ACTION A_DALICmdSetMinLevel_Input:
	IF emod = E_DALIAddressType.Group THEN
		byAddr		:= byGrpAdr;
		eAddrType	:= E_DALIAddressType.Group;
	ELSIF emod = E_DALIAddressType.Short THEN
		byAddr		:= byShrtAdr;
		eAddrType	:= E_DALIAddressType.Short;
	END_IF


	bActionBusy	:= TRUE;

	fbSetMinLevel(
		bError=> , 
		ipResultMessage=> , 
		bStart:= TRUE, 
		nAddress:= byAddr , 
		eAddressType:= eAddrType , 
		eCommandPriority:=Tc3_DALI.E_DALICommandPriority.Middle , 
		bBusy=> , 
		nMinLevel:= byDTR);
	

	IF (NOT fbSetMinLevel.bBusy) THEN
		IF fbSetMinLevel.bError THEN
			bErr := TRUE;
			nErrorId := fbSetMinLevel.ipResultMessage.nEventId;
		END_IF
		bActionBusy		:= FALSE;
		fbSetMinLevel(bStart:= FALSE);
	END_IF
END_ACTION

ACTION A_DALICmdStepDown:
	IF emod = E_DALIAddressType.Group THEN
		byAddr		:= byGrpAdr;
		eAddrType	:= E_DALIAddressType.Group;
	ELSIF emod = E_DALIAddressType.Short THEN
		byAddr		:= byShrtAdr;
		eAddrType	:= E_DALIAddressType.Short;
	END_IF

	bActionBusy	:= TRUE;

	fbStepDown(
		bError=> , 
		ipResultMessage=> , 
		bStart:= TRUE, 
		nAddress:=byAddr , 
		eAddressType:= eAddrType, 
		eCommandPriority:= E_DALICommandPriority.Middle, 
		bBusy=> );


	IF NOT fbStepDown.bBusy	THEN
		IF	fbStepDown.bError	THEN
			bErr     	:= TRUE;
		END_IF
		bActionBusy		:= FALSE;
		fbStepDown(bStart:= FALSE );
	END_IF
END_ACTION

ACTION A_DALICmdStepUp:
	IF emod = E_DALIAddressType.Group THEN
		byAddr		:= byGrpAdr;
		eAddrType	:= E_DALIAddressType.Group;
	ELSIF emod = E_DALIAddressType.Short THEN
		byAddr		:= byShrtAdr;
		eAddrType	:= E_DALIAddressType.Short;
	END_IF


	bActionBusy	:= TRUE;

	fbStepUp(
		bError=> , 
		ipResultMessage=> , 
		bStart:= TRUE, 
		nAddress:=byAddr , 
		eAddressType:=eAddrType , 
		eCommandPriority:= E_DALICommandPriority.Middle, 
		bBusy=> );


	IF NOT fbStepUp.bBusy	THEN
		IF	fbStepUp.bError	THEN
			bErr     	:= TRUE;
			nErrorId := fbStepUp.ipResultMessage.nEventId;

		END_IF
		bActionBusy		:= FALSE;
		fbStepUp(bStart:= FALSE);
	END_IF
END_ACTION

ACTION A_DALICmdUp:
	IF emod = E_DALIAddressType.Group THEN
		byAddr		:= byGrpAdr;
		eAddrType	:= E_DALIAddressType.Group;
	ELSIF emod = E_DALIAddressType.Short THEN
		byAddr		:= byShrtAdr;
		eAddrType	:= E_DALIAddressType.Short;
	END_IF

	bActionBusy	:= TRUE;

	fbUp(
		bError=> , 
		ipResultMessage=> , 
		bStart:= TRUE , 
		nAddress:=byAddr , 
		eAddressType:=eAddrType , 
		eCommandPriority:= E_DALICommandPriority.High, 
		bBusy=> );

	IF NOT fbUp.bBusy	THEN
		IF	fbUp.bError	THEN
			bErr     	:= TRUE;
			nErrorId := fbUp.ipResultMessage.nEventId;
		END_IF
		bActionBusy		:= FALSE;
		fbUp(bStart:= FALSE );
	END_IF
END_ACTION

ACTION A_ResetRoutine:
	tonSeqTimer(IN:=FALSE);
	tonDimRepeat(IN:=FALSE);

	bErr     	:= FALSE;
	nErrorId 	:= 0;


	fbUp						(bStart:= FALSE );
	fbDwn						(bStart:= FALSE );
	fbOff						(bStart:= FALSE );
	fbRecallMaxLevel			(bStart:= FALSE );
	fbRecallMinLevel			(bStart:= FALSE );
	fbDirectArcPowerControl		(bStart:= FALSE );
	fbStepUp					(bStart:= FALSE );
	fbStepDown					(bStart:= FALSE );
	fbQueryActualLevel			(bStart:= FALSE );
	fbSetFadeRate				(bStart:= FALSE );
	fbSetFadeTime				(bStart:= FALSE );
	fbQueryPhysicalMinLevel		(bStart:= FALSE );
	fbSetMinLevel				(bStart:= FALSE );
	fbQueryMinLevel				(bStart:= FALSE );
	fbSetMaxLevel				(bStart:= FALSE );
END_ACTION

{attribute 'monitoring' := 'call'}
PROPERTY ipDALICommunication : Tc3_DALI.I_DALICommunication
GET
ipDALICommunication := THIS^.ipCommunication;
END_GET
SET
THIS^.ipCommunicationPreset := ipDALICommunication;
END_SET
END_PROPERTY

//| Apply the perset value of IpCommunication if available
//| Return codes:
//|   FALSE: no peset value available
//|   TRUE: has taken the preset value
{attribute 'hide'}
METHOD PRIVATE TrySetCommunication : BOOL
VAR_INPUT
END_VAR
IF ((THIS^.ipCommunication <> THIS^.ipCommunicationPreset) AND (THIS^.ipCommunicationPreset <> 0)) THEN
	THIS^.ipCommunication := THIS^.ipCommunicationPreset;
	THIS^.fbUp.ipDALICommunication := THIS^.ipCommunication;
	THIS^.fbDwn.ipDALICommunication := THIS^.ipCommunication;
	THIS^.fbOff.ipDALICommunication := THIS^.ipCommunication;
	THIS^.fbRecallMaxLevel.ipDALICommunication := THIS^.ipCommunication;
	THIS^.fbRecallMinLevel.ipDALICommunication := THIS^.ipCommunication;
	THIS^.fbDirectArcPowerControl.ipDALICommunication := THIS^.ipCommunication;
	THIS^.fbStepUp.ipDALICommunication := THIS^.ipCommunication;	
	THIS^.fbStepDown.ipDALICommunication := THIS^.ipCommunication;
	THIS^.fbQueryActualLevel.ipDALICommunication := THIS^.ipCommunication;	
	THIS^.fbSetFadeRate.ipDALICommunication := THIS^.ipCommunication;
	THIS^.fbSetFadeTime.ipDALICommunication := THIS^.ipCommunication;
	THIS^.fbSetMaxLevel.ipDALICommunication := THIS^.ipCommunication;
	THIS^.fbSetMinLevel.ipDALICommunication := THIS^.ipCommunication;
	THIS^.fbQueryMinLevel.ipDALICommunication := THIS^.ipCommunication;	
	THIS^.fbQueryMaxLevel.ipDALICommunication := THIS^.ipCommunication;
	THIS^.fbQueryPhysicalMinLevel.ipDALICommunication := THIS^.ipCommunication;
	THIS^.fbQueryActualLevelBackgound.ipDALICommunication := THIS^.ipCommunication;
	THIS^.fbQueryStatusBackground.ipDALICommunication := THIS^.ipCommunication;
	TrySetCommunication := TRUE;
ELSE
	TrySetCommunication := FALSE;
END_IF
END_METHOD

END_FUNCTION_BLOCK

// POUs/DALI/Operators/FB_BA_ValTrigF
///Trigger-setting of a value, when it leaves a specific hysteresis
FUNCTION_BLOCK FB_BA_ValTrigF
VAR_INPUT
	bEn			: BOOL;		(* Enable *)
	bRetrig		: BOOL;		(* Retrigger - send bSet for one cycle *)
	fIn		: REAL;	(* Input signal *)
	fHys		: REAL;	(* Signal Hysteresis *)
END_VAR
VAR_OUTPUT
	fOut		: REAL;
	bSet		: BOOL;
END_VAR
VAR
	bInit		: BOOL;
	rtRetrig1	: R_TRIG;
	rtRetrig2	: R_TRIG;
	fLimUp		: REAL;
	fLimDwn		: REAL;
	uiStep		: UINT;
END_VAR

IF NOT bInit	THEN
	fLimUp	:= fIn+fHys/2;
	fLimDwn:= fIn-fHys/2;
	fOut	:= fIn;
	bInit	:= TRUE;
END_IF

rtRetrig1(CLK:=bEn); 		(*Retrigger both at retrigger-command and at beginning of enable*)
rtRetrig2(CLK:=bRetrig); (*Retrigger both at retrigger-command and at beginning of enable*)

CASE uiStep OF
0: (*Idle*)
	bSet:=FALSE;
	IF (fIn>=fLimUp)OR(fIn<=fLimDwn) OR rtRetrig1.Q	OR rtRetrig2.Q	THEN
		uiStep	:= 10;
	END_IF
	IF NOT bEn	THEN
		uiStep	:= 0;
	END_IF

10:
	fLimUp	:= fIn+fHys/2;
	fLimDwn	:= fIn-fHys/2;
	fOut	:= fIn;
	bSet	:= TRUE;
	uiStep 	:= 0;
END_CASE

END_FUNCTION_BLOCK

// POUs/DALI/Ballast/FB_DALILgtActr_Simple
FUNCTION_BLOCK FB_DALILgtActr_Simple  (* V1.1 dfgdfgdfgdfgdfgfzxcv *)
VAR_INPUT
	byShrtAdr				: BYTE;
	byGrpAdr				: BYTE;
	eMod					: E_DALIAddressType:= E_DALIAddressType.Group;
	fSttupCtrlVal			: REAL;
	fLgtOffset				: REAL;
	uiBlinkTi				: UINT;
	uiOffDly				: UINT;
	uiPollActLgtLvl			: UINT;
	bReInit					: BOOL;
	stLgtCmd				: ST_LgtCmd;
	DALI_LINE_NUM			: BYTE;
END_VAR
VAR_OUTPUT
	fActlLgtLvl				: REAL;
	byActlLgtLvl			: BYTE;
	bLgt					: BOOL;
	fActlMinCtrlVal			: REAL;
	bMinCtrlValRchd 		: BOOL;
	fActlMaxCtrlVal			: REAL;
	bMaxCtrlValRchd 		: BOOL;
	fRstVal					: REAL;
	eActlFadeTime			: E_DALIFadeTime;
	eActlFadeRate			: E_DALIFadeRate;
	byPhysMinVal			: BYTE;
	byActlMinCtrlVal		: BYTE;
	byActlMaxCtrlVal		: BYTE;
	bInitDevice				: BOOL;
	bBlinkSeqStarted 		: BOOL;
	bActionBusy				: BOOL;
	bErr     				: BOOL;
	nErrorId				: UDINT;
	byDALIDevSta			: BYTE;
END_VAR
VAR
	ipCommunication					: I_DALICommunication;
	ipCommunicationPreset			: I_DALICommunication;

	bInit					: BOOL;
	bBusy					: BOOL;
	bRstErr					: BOOL;
	rtReInit				: R_TRIG;
	bReactCmdSt				: BOOL;
	byAddr					: BYTE;
	eAddrType				: E_DALIAddressType;
	byArcPowerLevel			: BYTE;
	byDTR					: BYTE;
	uiCmdStep				: UINT;

	bDimUp					: BOOL;
	bDimDwn					: BOOL;
	bSetMinValInput			: BOOL;	(*Änderung MinVal über Bausteineingang*)
	bSetMaxValInput			: BOOL;	(*Änderung MaxVal über Bausteineingang*)
	bySetMinValInput		: BYTE;
	bySetMaxValInput		: BYTE;
	bSetMinValCmdSt			: BOOL;	(*Änderung MinVal über Kommandostruktur*)
	bSetMaxValCmdSt			: BOOL;	(*Änderung MaxVal über Kommandostruktur*)
	bySetMinValCmdSt		: BYTE;
	bySetMaxValCmdSt		: BYTE;
	byRstVal				: BYTE;
	bySttupCtrlVal			: BYTE;
	rtInitDevice			: R_TRIG;
	rtOff					: R_TRIG;
	rtClMinCtrlVal			: R_TRIG;
	rtClMaxCtrlVal			: R_TRIG;
	rtClOnVal				: R_TRIG;
	rtClRstVal				: R_TRIG;
	rtSetCtrlValDct			: R_TRIG;
	rtChgMaxCtrlVal			: R_TRIG;
	rtChgMinCtrlVal			: R_TRIG;
	rtStpUp							: R_TRIG;
	rtStpDwn						: R_TRIG;
	rtRmp							: R_TRIG;
	tonSeqTimer						: TON;
	tonDimRepeat					: TON;
	fbUp							: FB_DALI102Up(0);
	fbDwn							: FB_DALI102Down(0);
	fbOff							: FB_DALI102Off(0);
	fbRecallMaxLevel				: FB_DALI102RecallMaxLevel(0);
	fbRecallMinLevel				: FB_DALI102RecallMinLevel(0);
	fbDirectArcPowerControl			: FB_DALI102DirectArcPowerControl(0);
	fbStepUp						: FB_DALI102StepUp(0);
	fbStepDown						: FB_DALI102StepDown(0);
	fbQueryActualLevel				: FB_DALI102QueryActualLevel(0);
	fbQueryMinLevel					: FB_DALI102QueryMinLevel(0);
	fbQueryMaxLevel					: FB_DALI102QueryMaxLevel(0);
	fbQueryPhysicalMinLevel			: FB_DALI102QueryPhysicalMinimum(0);
	fbQueryActualLevelBackgound		: FB_DALI102QueryActualLevel(0);
	fbQueryStatusBackground			: FB_DALI102QueryStatus(0);
	fbSendValue						: FB_BA_ValTrigf;
	fbReTrigSend0					: R_TRIG;
	nStepQueryActualLevel			: UINT;
	tonCycleActualLevelMasterDev	: TON;
	bSetRetry						: BOOL;
	fbTimeOut						: TON;
	byActlFadeTime					: BYTE;
	fbGETCURTASKINDEX				: GETCURTASKINDEX;
	nCurrentIdx						: BYTE;
	nCycleTimeInMS					: UDINT;
	nCycleCountSP					: UDINT;
	nActualCount					: UDINT:= 1;
END_VAR
VAR_IN_OUT
END_VAR



(* For checking which task the FB are called*)
fbGETCURTASKINDEX(index=>nCurrentIdx );
nCycleTimeInMS:= (_TaskInfo[nCurrentIdx].CycleTime/10000);
IF nCycleTimeInMS > 0 THEN	(*nCycleCountSP are only calculated if nCycleTimeInMS are larger than 0*)
	nCycleCountSP:= (200 / nCycleTimeInMS) ; (* 200 are the target time between 2 UP/Down cmd*)
END_IF

{region "initialize the outputs"}
IF (NOT bInit) THEN
	THIS^.TrySetCommunication();		 
	bBusy := TRUE;
	nErrorId := 0;
	bErr := FALSE;
	bInit := TRUE;
END_IF
{endregion}


{region "check parameters"}
IF (ipCommunication = 0) THEN
	bErr := TRUE;
	nErrorId := TC_EVENTS.TcDALIEventClass.TheInterfaceToTheCommunicationBufferIsNotInitialized.nEventId;
	uiCmdStep := 0;
END_IF
IF ((eMod <> E_DALIAddressType.Short) AND (eMod <> E_DALIAddressType.Group) AND (eMod <> E_DALIAddressType.Broadcast) AND (eMod <> E_DALIAddressType.BroadcastUnaddr)) THEN
	bErr := TRUE;
	nErrorId := TC_EVENTS.TcDALIEventClass.ParameterAddressTypeLiesOutsideOfTheValidRange.nEventId;
	uiCmdStep := 0;
END_IF
IF ((eMod = E_DALIAddressType.Short) AND (byShrtAdr > 63)) THEN
	bErr := TRUE;
	nErrorId := TC_EVENTS.TcDALIEventClass.ParameterAddressIsAShortAddressAndLiesOutsideOfTheValidRange.nEventId;
	uiCmdStep := 0;
END_IF
IF ((eMod = E_DALIAddressType.Group) AND (byGrpAdr > 15)) THEN
	bErr := TRUE;
	nErrorId := TC_EVENTS.TcDALIEventClass.ParameterAddressIsAGroupAddressAndLiesOutsideOfTheValidRange.nEventId;
	uiCmdStep := 0;
END_IF
IF (byShrtAdr > 63) THEN
	bErr := TRUE;
	nErrorId := 16#8000; // custom error code: Parameter byShrtAdr lies outside of the valid range
	uiCmdStep := 0;
END_IF
	
IF (byGrpAdr > 15) THEN
	bErr := TRUE;
	nErrorId := 16#8001; // custom error code: Parameter byGrpAdr lies outside of the valid range
	uiCmdStep := 0;
END_IF
{endregion}

(*	bRstErr ist ein Fehlermerker: wenn vorher über Fehler, s.o. herausgesprungen wurde und nun "alles gut" ist,
dann hier Fehler einmalig zurücksetzen, damit im weiteren Verlauf die Warnmeldungen sichtbar werden können*)
IF	bRstErr  THEN
		bRstErr    	:= FALSE;
		bErr     	:= FALSE;
END_IF


(* + + + + + + + + + + + + + + + + + + + + + + + + + + + + + + + + + + + + + + + + + + + + *)
(*In den DALI-Ausführungsaktionen ist jedoch zur Sicherheit noch ein RETURN-Aussprung*)
IF (eMod=E_DALIAddressType.Short)	THEN
	bReactCmdSt:=FALSE;
ELSE
	bReactCmdSt:=TRUE;
END_IF

(* + + + + + + + + + + + + + + + + + + + + + + + + + + + + + + + + + + + + + + + + + + + + *)
(*Init *)
rtReInit	 (CLK:=bReInit);
IF bReInit	THEN
	bInit:=FALSE;
END_IF

IF NOT bInit	THEN
	rtInitDevice			(CLK:=FALSE);
	bInitDevice			:= TRUE;

	bInit					:= TRUE;
	tonDimRepeat		(PT:=t#200ms);

	IF fSttupCtrlVal < 0.0	 THEN
		bySttupCtrlVal	:= 0;
	ELSIF	fSttupCtrlVal > 100.0	 THEN
		bySttupCtrlVal	:= 254;
	ELSE
		bySttupCtrlVal	:= LREAL_TO_BYTE(F_fDALICurve(fSttupCtrlVal));
	END_IF
END_IF

rtInitDevice (CLK:=bInitDevice);

(*Removed in Simple version, Other FB needed for setup ballast - HMB 14/12-2021*)
(*

(* + + + + + + + + + + + + + + + + + + + + + + + + + + + + + + + + + + + + + + + + + + + + *)
(*Change DimTime/FadeRate über Bausteineingang*)
IF	(uiDimTi<>uiDimTi_SV) OR rtInitDevice.Q THEN
	A_DimTimeToFadeRate;
	uiDimTi_SV	:= uiDimTi;
	IF NOT rtInitDevice.Q	THEN
		bSetFadeRate	:= TRUE;
	END_IF
END_IF

(* + + + + + + + + + + + + + + + + + + + + + + + + + + + + + + + + + + + + + + + + + + + + *)
(*Change Min-/MaxCtrlVal über Bausteineingang*)

IF	(lrMinCtrlVal<>lrMinCtrlVal_SV) OR rtInitDevice.Q THEN
	lrMinCtrlVal_SV		:= lrMinCtrlVal;
	IF 		lrMinCtrlVal < 0.0		 THEN
		bySetMinValInput	:= 0;
	ELSIF	lrMinCtrlVal > 100.0	 THEN
		bySetMinValInput	:= 254;
	ELSE
		bySetMinValInput	:= LREAL_TO_BYTE(lrMinCtrlVal*2.54);
	END_IF
	IF NOT rtInitDevice.Q	THEN
		bSetMinValInput	:= TRUE;
	END_IF
END_IF

IF	(lrMaxCtrlVal<>lrMaxCtrlVal_SV) OR rtInitDevice.Q THEN
	lrMaxCtrlVal_SV		:= lrMaxCtrlVal;
	IF 		lrMaxCtrlVal < 0.0		 THEN
		bySetMaxValInput	:= 0;
	ELSIF	lrMaxCtrlVal > 100.0	 THEN
		bySetMaxValInput	:= 254;
	ELSE
		bySetMaxValInput	:= LREAL_TO_BYTE(lrMaxCtrlVal*2.54);
	END_IF
	IF NOT rtInitDevice.Q	THEN
		bSetMaxValInput	:= TRUE;
	END_IF
END_IF


(* + + + + + + + + + + + + + + + + + + + + + + + + + + + + + + + + + + + + + + + + + + + + *)
(*Change Min-/MaxCtrlVal über Kommandostruktur*)
rtChgMinCtrlVal	(CLK:= stLgtCmd.bChgMinCtrlVal);
rtChgMaxCtrlVal	(CLK:= stLgtCmd.bChgMaxCtrlVal);

IF 	rtChgMinCtrlVal.Q	AND bReactCmdSt			THEN
	IF 		stLgtCmd.lrChgMinCtrlVal < 0.0		 THEN
		bySetMinValCmdSt	:= 0;
	ELSIF	stLgtCmd.lrChgMinCtrlVal > 100.0	 THEN
		bySetMinValCmdSt	:= 254;
	ELSE
		bySetMinValCmdSt	:= LREAL_TO_BYTE(stLgtCmd.lrChgMinCtrlVal*2.54);
	END_IF
	bSetMinValCmdSt	:= TRUE;
END_IF

IF 	rtChgMaxCtrlVal.Q	AND bReactCmdSt			THEN
	IF 		stLgtCmd.lrChgMaxCtrlVal < 0.0		 THEN
		bySetMaxValCmdSt	:= 0;
	ELSIF	stLgtCmd.lrChgMaxCtrlVal > 100.0	 THEN
		bySetMaxValCmdSt	:= 254;
	ELSE
		bySetMaxValCmdSt	:= LREAL_TO_BYTE(stLgtCmd.lrChgMaxCtrlVal*2.54);
	END_IF
	bSetMaxValCmdSt	:= TRUE;
END_IF
*)

fbSendValue(bEn:= TRUE, bRetrig:= , fIn:= stLgtCmd.fSetCtrlValDct, fHys:= 0.1);

IF bMinCtrlValRchd AND stLgtCmd.fSetCtrlValDct = 0 THEN
	fbReTrigSend0(CLK:=TRUE , Q=> );
ELSE
	fbReTrigSend0(CLK:=FALSE , Q=> );
END_IF

(* + + + + + + + + + + + + + + + + + + + + + + + + + + + + + + + + + + + + + + + + + + + + *)
(* Flankenbildung und Verriegelung der Schalt- und Dimmbefehle *)
rtOff			(CLK:=stLgtCmd.bOff OR fbReTrigSend0.Q);
rtClMinCtrlVal	(CLK:=stLgtCmd.bClMinCtrlVal);
rtClMaxCtrlVal	(CLK:=stLgtCmd.bClMaxCtrlVal);
rtClOnVal		(CLK:=stLgtCmd.bClOnVal);
rtClRstVal		(CLK:=stLgtCmd.bClRstVal);
rtSetCtrlValDct	(CLK:=stLgtCmd.bSetCtrlValDct OR fbSendValue.bSet);
rtStpUp			(CLK:=stLgtCmd.bStpUp);
rtStpDwn		(CLK:=stLgtCmd.bStpDwn);

bDimUp			:= stLgtCmd.bDimUp;
bDimDwn			:= stLgtCmd.bDimDwn;

(* + + + + + + + + + + + + + + + + + + + + + + + + + + + + + + + + + + + + + + + + + + + + *)
(* Priorisierung aller Befehle und Schrittzuweisung *)
IF NOT bBusy	THEN
	IF			rtInitDevice.Q		THEN
				bBusy := TRUE;
								A_ResetRoutine();
				uiCmdStep:=1030;	(*Jump over write to ballast, else set back to step 1000*)
	ELSIF	bDimUp				AND NOT bMaxCtrlValRchd THEN
				bBusy := TRUE;
				A_ResetRoutine();
				uiCmdStep:=10;
	ELSIF	bDimDwn				AND NOT bMinCtrlValRchd THEN
				bBusy := TRUE;
				A_ResetRoutine();
				uiCmdStep:=20;
	ELSIF	rtOff.Q				THEN
				bBusy := TRUE;
				A_ResetRoutine();
				uiCmdStep:=30;
	ELSIF	rtClMinCtrlVal.Q	THEN
				bBusy := TRUE;
				A_ResetRoutine();
				uiCmdStep:=40;
	ELSIF	rtClMaxCtrlVal.Q	THEN
				bBusy := TRUE;
				A_ResetRoutine();
				uiCmdStep:=50;
	ELSIF	rtClOnVal.Q	THEN
				bBusy := TRUE;
				A_ResetRoutine();
				uiCmdStep:=60;
	ELSIF	rtClRstVal.Q		THEN
				bBusy := TRUE;
				A_ResetRoutine();
				uiCmdStep:=70;
	ELSIF	rtSetCtrlValDct.Q	THEN
				bBusy := TRUE;
				A_ResetRoutine();
				uiCmdStep:=80;
	ELSIF	rtStpUp.Q			AND NOT bMaxCtrlValRchd THEN
				bBusy := TRUE;
				A_ResetRoutine();
				uiCmdStep:=90;
	ELSIF	rtStpDwn.Q			AND NOT bMinCtrlValRchd THEN
				bBusy := TRUE;
				A_ResetRoutine();
				uiCmdStep:=100;
	END_IF
END_IF

(* + + + + + + + + + + + + + + + + + + + + + + + + + + + + + + + + + + + + + + + + + + + + *)
(*Kommandoausgabe*)
CASE uiCmdStep OF

0: (*Idle*)
	bInitDevice := FALSE;
	bBusy := FALSE;


(* - - - - - - - - - - - - - - - - - - - - - - - - *)
10:(*Dim Up*)
	bBlinkSeqStarted := FALSE;
(*	tonDimRepeat	(IN:=TRUE); *)  (*Disabled for at teste om Up cmd kommer hurtigere ved at tælle skan, istedet for timer*)
	nActualCount:= 1;
		A_DALICmdUp();
	IF NOT bActionBusy	THEN
		uiCmdStep:= 11;
	END_IF

11:(*Ende Wartezeit 200ms abwarten*)

(*Disablet to be more precise in case of long scantimes in the task - HMB 13/12-2021*)
(*	tonDimRepeat();
	IF tonDimRepeat.Q THEN
		tonDimRepeat(IN:= FALSE);
		IF bDimUp		THEN
			uiCmdStep:=10;
		ELSE
			uiCmdStep:=12;
		END_IF
	END_IF
*)
	(* Added to see if 200ms can be reached with this scan count*)
	IF nActualCount <= nCycleCountSP THEN
		nActualCount := nActualCount + 1;
		IF nActualCount >=nCycleCountSP THEN
			nActualCount:=1;
			IF bDimUp		THEN
				uiCmdStep:=10;
			ELSE
				uiCmdStep:=12;
			END_IF
		END_IF
	END_IF


12: (*Lichtabfrage wenn fertig*)
		A_DALICmdQueryActualLevel();
	IF NOT bActionBusy	THEN
		byActlLgtLvl	:= fbQueryActualLevel.nActualLevel;
		uiCmdStep		:= 0;
	END_IF

(* - - - - - - - - - - - - - - - - - - - - - - - - *)
20:(*Dim Down*)
	bBlinkSeqStarted := FALSE;
(*	tonDimRepeat	(IN:=TRUE); *)  (*Disabled for at teste om Up cmd kommer hurtigere ved at tælle skan, istedet for timer*)
	nActualCount:= 1;
		A_DALICmdDown();
	IF NOT bActionBusy	THEN
		uiCmdStep:= 21;
	END_IF

21:(*Ende Wartezeit 200ms abwarten*)
(*Disablet to be more precise in case of long scantimes in the task - HMB 13/12-2021*)
(*	tonDimRepeat();
	IF tonDimRepeat.Q THEN
		tonDimRepeat(IN:= FALSE);
		IF bDimDwn		THEN
			uiCmdStep:=20;
		ELSE
			uiCmdStep:=22;
		END_IF
	END_IF
*)
	IF nActualCount <= nCycleCountSP THEN
		nActualCount := nActualCount + 1;
		IF nActualCount >=nCycleCountSP THEN
			nActualCount:= 1;
			IF bDimDwn	THEN
				uiCmdStep:=20;
			ELSE
				uiCmdStep:=22;
			END_IF
		END_IF
	END_IF

22: (*Lichtabfrage wenn fertig*)
		A_DALICmdQueryActualLevel();
	IF NOT bActionBusy	THEN
		byActlLgtLvl	:= fbQueryActualLevel.nActualLevel;
		uiCmdStep		:= 0;
	END_IF

(* - - - - - - - - - - - - - - - - - - - - - - - - *)
30:(*Off*)
		A_DALICmdOff();
	IF NOT bActionBusy	THEN
		byActlLgtLvl	:=0;
		IF (uiOffDly<>0) AND NOT bBlinkSeqStarted AND NOT bErr	THEN
			uiCmdStep:=500;
		ELSE
			bBlinkSeqStarted := FALSE;
			uiCmdStep:= 0;
		END_IF
	END_IF

(* - - - - - - - - - - - - - - - - - - - - - - - - *)
40:(*Call MinCtrlVal*)
	bBlinkSeqStarted := FALSE;
		A_DALICmdRecallMinLevel();
	IF NOT bActionBusy	THEN
		byActlLgtLvl:=byActlMinCtrlVal;
		uiCmdStep:= 0;
	END_IF

(* - - - - - - - - - - - - - - - - - - - - - - - - *)
50:(*Call MaxCtrlVal*)
	bBlinkSeqStarted := FALSE;
		A_DALICmdRecallMaxLevel();
	IF NOT bActionBusy	THEN
		byActlLgtLvl:=byActlMaxCtrlVal;
		uiCmdStep:= 0;
	END_IF

(* - - - - - - - - - - - - - - - - - - - - - - - - *)
60:(*Call OnVal*)
	(*Limitation is not to be left to the electrical device -> the output of the actual value would be left to the background-polling only*)
	IF ((stLgtCmd.lrOnVal)>=fActlMaxCtrlVal)	THEN
		byArcPowerLevel:=byActlMaxCtrlVal;
	ELSIF ((stLgtCmd.lrOnVal)<=0.0)	THEN
		byArcPowerLevel:=0;
	ELSIF ((stLgtCmd.lrOnVal)<=fActlMinCtrlVal)	THEN
		byArcPowerLevel:=byActlMinCtrlVal;
	ELSE
		byArcPowerLevel:=LREAL_TO_BYTE((stLgtCmd.lrOnVal)*2.54);
	END_IF

		A_DALICmdDirectArcPowerControl();
	IF NOT bActionBusy	THEN
		byActlLgtLvl:=byRstVal;
		uiCmdStep:= 0;
	END_IF

(* - - - - - - - - - - - - - - - - - - - - - - - - *)
70:(*Call ResetVal*)
	bBlinkSeqStarted := FALSE;
	byArcPowerLevel	:= byRstVal;
		A_DALICmdDirectArcPowerControl();
	IF NOT bActionBusy	THEN
		byActlLgtLvl:=byRstVal;
		uiCmdStep:= 0;
	END_IF

(* - - - - - - - - - - - - - - - - - - - - - - - - *)
80:(*Set Control value directly*)
	(*Limitation is not to be left to the electrical device -> the output of the actual value would be left to the background-polling only*)
	byArcPowerLevel:= LIMIT(0,LREAL_TO_BYTE(F_fDALICurve(stLgtCmd.fSetCtrlValDct+ fLgtOffset)),254);
	A_DALICmdDirectArcPowerControl();
	IF NOT bActionBusy	THEN
(*		byActlLgtLvl:=byArcPowerLevel;*)
		IF (byActlLgtLvl=0) AND (uiOffDly<>0) AND NOT bBlinkSeqStarted AND NOT bErr	THEN
			uiCmdStep:=500;
		ELSE
			bBlinkSeqStarted := FALSE;
			uiCmdStep:= 0;
		END_IF
	END_IF

(* - - - - - - - - - - - - - - - - - - - - - - - - *)
90:(*Step Up*)
	bBlinkSeqStarted := FALSE;
		A_DALICmdStepUp();
	IF NOT bActionBusy	THEN
		byActlLgtLvl:=byActlLgtLvl+1;
		IF	byActlLgtLvl>byActlMaxCtrlVal	THEN
			byActlLgtLvl:=byActlMaxCtrlVal;
		END_IF
		uiCmdStep:= 0;
	END_IF

(* - - - - - - - - - - - - - - - - - - - - - - - - *)
100:(*Step Down*)
	bBlinkSeqStarted := FALSE;
		A_DALICmdStepDown();
	IF NOT bActionBusy	THEN
		byActlLgtLvl:=byActlLgtLvl-1;
		IF	byActlLgtLvl<byActlMinCtrlVal	THEN
			byActlLgtLvl:=byActlMinCtrlVal;
		END_IF
		uiCmdStep:= 0;
	END_IF


(* - - - - - - - - - - - - - - - - - - - - - - - - *)
(*ZUR SICHERHEIT: ABFRAGE NACH PARAMETRIERUNG*)
350:(*Query Min Level*)
	A_DALICmdQueryMinLevel();
	IF NOT bActionBusy	THEN
		IF bErr	THEN
			uiCmdStep:= 0;
		ELSE
			uiCmdStep:= 351;
		END_IF
	END_IF
	byActlMinCtrlVal:=fbQueryMinLevel.nMinLevel;
	fActlMinCtrlVal := LIMIT(0,LREAL_TO_BYTE(F_fDALICurve(byActlMinCtrlVal)), 254);

351:(*Query Max Level*)
	A_DALICmdQueryMaxLevel();
	IF NOT bActionBusy	THEN
		IF bErr	THEN
			uiCmdStep:= 0;
		ELSE
			uiCmdStep:= 352;
		END_IF
	END_IF
	byActlMaxCtrlVal:=fbQueryMaxLevel.nMaxLevel;
	fActlMaxCtrlVal := LIMIT(0,LREAL_TO_BYTE(F_fDALICurve(byActlMaxCtrlVal)), 254);

352: (*Lichtabfrage wenn fertig*)
		A_DALICmdQueryActualLevel();
	IF NOT bActionBusy	THEN
		byActlLgtLvl	:= fbQueryActualLevel.nActualLevel;
		uiCmdStep		:= 0;
	END_IF


(* - - - - - - - - - - - - - - - - - - - - - - - - *)
(*Ausschalt-Blinksequenz*)
500: (*Lampe ist bereits aus -> Wartezeit Blinktime*)
	bBusy				:= FALSE;	(*Blinksequenz soll unterbrechbar sein*)
	bBlinkSeqStarted	:= TRUE;
	tonSeqTimer			(IN:= TRUE, PT:=UDINT_TO_TIME(uiBlinkTi*1000));

	IF tonSeqTimer.Q	THEN
		bBusy := TRUE;	(*Verriegelung Kommandoannahme*)
		tonSeqTimer(IN:=FALSE);
		uiCmdStep:= 505;
	END_IF

505: (*Zurück auf ürsprünglich gespeicherten Wert*)
	byArcPowerLevel	:= byRstVal;
		A_DALICmdDirectArcPowerControl();
	IF NOT bActionBusy	THEN
		byActlLgtLvl := byRstVal;
		bBusy:= FALSE;	(*Blinksequenz soll wieder unterbrechbar sein*)
		IF bErr	THEN
			uiCmdStep:= 0;
		ELSE
			uiCmdStep:= 510;
		END_IF
	END_IF

510:(*Wartezeit Off-Delaytime*)
	tonSeqTimer(IN:= TRUE, PT:=UDINT_TO_TIME(uiOffDly*1000));
	IF tonSeqTimer.Q THEN
		bBusy := TRUE;	(*Verriegelung Kommandoannahme*)
		tonSeqTimer(IN:=FALSE);
		uiCmdStep:= 515;
	END_IF

515:(*Off*)
		A_DALICmdOff();
	IF NOT bActionBusy	THEN
		byActlLgtLvl		:= 0;
		bBlinkSeqStarted	:= FALSE;
		bBusy				:= FALSE;
		uiCmdStep			:= 0;
	END_IF

(* - - - - - - - - - - - - - - - - - - - - - - - - *)
(*Init Device-Routine*)

1000: (*Wait fort free DT8*)
	IF NOT arrbBlockDTR[DALI_LINE_NUM] THEN
		uiCmdStep:= 1030;
		arrbBlockDTR[DALI_LINE_NUM]:= FALSE;
	END_IF


1030:(*Query physical Min Level*)
		A_DALICmdQueryPhysicalMinLevel();
	IF NOT bActionBusy	THEN
		IF bErr	THEN
			uiCmdStep:= 0;
			arrbBlockDTR[DALI_LINE_NUM]:=FALSE;
		ELSE
			uiCmdStep:= 1035;
		END_IF
	END_IF
	byPhysMinVal:=fbQueryPhysicalMinLevel.nPhysicalMinimum;

1035:(*Query Min Level*)
		A_DALICmdQueryMinLevel();
	IF NOT bActionBusy	THEN
		IF bErr	THEN
			uiCmdStep:= 0;
			arrbBlockDTR[DALI_LINE_NUM]:=FALSE;
		ELSE
			uiCmdStep:= 1040;
		END_IF
	END_IF
	byActlMinCtrlVal:=fbQueryMinLevel.nMinLevel;
	fActlMinCtrlVal := LIMIT(0,LREAL_TO_BYTE(F_fDALICurve(byActlMinCtrlVal)), 254);

1040:(*Query Max Level*)
		A_DALICmdQueryMaxLevel();
	IF NOT bActionBusy	THEN
		IF bErr	THEN
			uiCmdStep:= 0;
			arrbBlockDTR[DALI_LINE_NUM]:=FALSE;
		ELSE
			uiCmdStep:= 1045;
		END_IF
	END_IF
	byActlMaxCtrlVal:=fbQueryMaxLevel.nMaxLevel;
	fActlMaxCtrlVal := LIMIT(0,LREAL_TO_BYTE(F_fDALICurve(byActlMaxCtrlVal)), 254);

1045:(*Call Startup-Level*)
	byArcPowerLevel	:= bySttupCtrlVal;
		A_DALICmdDirectArcPowerControl_Sttup();
	IF NOT bActionBusy	THEN
		uiCmdStep:= 1050;
	END_IF

1050: (*Lichtabfrage wenn fertig*)
		A_DALICmdQueryActualLevel();
	IF NOT bActionBusy	THEN
		byActlLgtLvl	:= fbQueryActualLevel.nActualLevel;
		uiCmdStep		:= 0;
		arrbBlockDTR[DALI_LINE_NUM]:=FALSE;
	END_IF

END_CASE

(*+ + + + + + + + + + + + + + + + + + + + + + + + + + + + + + + + + + + + + + + + + + + + + + + + +*)

IF ((uiPollActLgtLvl > 0) AND (nStepQueryActualLevel = 0) AND (bErr = FALSE)) THEN
	tonCycleActualLevelMasterDev(IN := TRUE, PT := UINT_TO_TIME(uiPollActLgtLvl*1000));
	IF (tonCycleActualLevelMasterDev.Q) THEN
		tonCycleActualLevelMasterDev(IN := FALSE);
		nStepQueryActualLevel := 10;
	END_IF
END_IF

CASE nStepQueryActualLevel OF
0:
	;
10:
	fbQueryActualLevelBackgound(
		bError=> , 
		ipResultMessage=> , 
		bStart:= TRUE, 
		nAddress:= byShrtAdr, 
		eAddressType:= E_DALIAddressType.Short, 
		eCommandPriority:=E_DALICommandPriority.Low , 
		bBusy=> , 
		nActualLevel=> );

	IF (NOT fbQueryActualLevelBackgound.bBusy) THEN
		IF (NOT fbQueryActualLevelBackgound.bError) THEN
			byActlLgtLvl := fbQueryActualLevelBackgound.nActualLevel;
		END_IF
		fbQueryActualLevelBackgound(bStart := FALSE);
		nStepQueryActualLevel := 20;
	END_IF

20:
	fbQueryStatusBackground(
		bError=> , 
		ipResultMessage=> , 
		bStart:= TRUE, 
		nAddress:= byShrtAdr, 
		eAddressType:= E_DALIAddressType.Short, 
		eCommandPriority:= E_DALICommandPriority.Low, 
		bBusy=> , 
		nStatus=> );

	IF (NOT fbQueryStatusBackground.bBusy) THEN
		IF (NOT fbQueryStatusBackground.bError) THEN
			byDALIDevSta := fbQueryStatusBackground.nStatus;
		END_IF
		fbQueryStatusBackground(bStart := FALSE);
		nStepQueryActualLevel := 0;
	END_IF
END_CASE

(* + + + + + + + + + + + + + + + + + + + + + + + + + + + + + + + + + + + + + + + + + + + + *)
(*Umrechnung des Lichtwertes lrActlLgtLvl und Speicherung des letzten Wertes vor Aus*)
bLgt			:= BYTE_TO_BOOL		(byActlLgtLvl);
(*lrActlLgtLvl	:= BYTE_TO_LREAL	(byActlLgtLvl)/2.54;*)
fActlLgtLvl	:= F_fDALICurveRev(BYTE_TO_REAL (byActlLgtLvl));

bMinCtrlValRchd:=(byActlLgtLvl=byActlMinCtrlVal);
bMaxCtrlValRchd:=(byActlLgtLvl=byActlMaxCtrlVal);

IF bLgt THEN
	byRstVal:= byActlLgtLvl;
	fRstVal := LIMIT(0,LREAL_TO_BYTE(F_fDALICurve(byActlLgtLvl)), 254);

END_IF

ACTION A_DALICmdDirectArcPowerControl:
	IF emod = E_DALIAddressType.Group THEN
		byAddr		:= byGrpAdr;
		eAddrType	:= E_DALIAddressType.Group;
	ELSIF emod = E_DALIAddressType.Short THEN
		byAddr		:= byShrtAdr;
		eAddrType	:= E_DALIAddressType.Short;
	END_IF


	bActionBusy	:= TRUE;

	fbDirectArcPowerControl(
		bError=> , 
		ipResultMessage=> , 
		bStart:=TRUE , 
		nAddress:= byAddr, 
		eAddressType:= eAddrType, 
		eCommandPriority:=Tc3_DALI.E_DALICommandPriority.Middle , 
		bBusy=> , 
		nArcPowerLevel:= byArcPowerLevel);

	IF NOT fbDirectArcPowerControl.bBusy	THEN
		IF	fbDirectArcPowerControl.bError	THEN
			bErr     	:= TRUE;
			nErrorId := fbDirectArcPowerControl.ipResultMessage.nEventId;
		END_IF
		byActlLgtLvl:=byArcPowerLevel;
		bActionBusy		:= FALSE;
		fbDirectArcPowerControl(bStart:= FALSE);
	END_IF
END_ACTION

ACTION A_DALICmdDirectArcPowerControl_Sttup:
	IF emod = E_DALIAddressType.Group THEN
		byAddr		:= byGrpAdr;
		eAddrType	:= E_DALIAddressType.Group;
	ELSIF emod = E_DALIAddressType.Short THEN
		byAddr		:= byShrtAdr;
		eAddrType	:= E_DALIAddressType.Short;
	END_IF

	bActionBusy	:= TRUE;

	fbDirectArcPowerControl(
		bError=> , 
		ipResultMessage=> , 
		bStart:=TRUE , 
		nAddress:= byAddr, 
		eAddressType:= eAddrType, 
		eCommandPriority:=Tc3_DALI.E_DALICommandPriority.Middle , 
		bBusy=> , 
		nArcPowerLevel:= byArcPowerLevel);	
	

	IF NOT fbDirectArcPowerControl.bBusy	THEN
		IF	fbDirectArcPowerControl.bError	THEN
			bErr     	:= TRUE;
			nErrorId := fbDirectArcPowerControl.ipResultMessage.nEventId;
		END_IF
		bActionBusy		:= FALSE;
		fbDirectArcPowerControl(bStart:= FALSE);
	END_IF
END_ACTION

ACTION A_DALICmdDown:
	IF emod = E_DALIAddressType.Group THEN
		byAddr		:= byGrpAdr;
		eAddrType	:= E_DALIAddressType.Group;
	ELSIF emod = E_DALIAddressType.Short THEN
		byAddr		:= byShrtAdr;
		eAddrType	:= E_DALIAddressType.Short;
	END_IF

	bActionBusy	:= TRUE;
	
	fbDwn(
		bError=> , 
		ipResultMessage=> , 
		bStart:= , 
		nAddress:= byAddr, 
		eAddressType:= eAddrType, 
		eCommandPriority:= Tc3_DALI.E_DALICommandPriority.High, 
		bBusy=> );
	
	
	IF NOT fbDwn.bBusy	THEN
		IF	fbDwn.bError	THEN
			bErr     	:= TRUE;
			nErrorId := fbDwn.ipResultMessage.nEventId;
		END_IF
		bActionBusy		:= FALSE;
		fbDwn(bStart:= FALSE);
	END_IF
END_ACTION

ACTION A_DALICmdOff:
	IF emod = E_DALIAddressType.Group THEN
		byAddr		:= byGrpAdr;
		eAddrType	:= E_DALIAddressType.Group;
	ELSIF emod = E_DALIAddressType.Short THEN
		byAddr		:= byShrtAdr;
		eAddrType	:= E_DALIAddressType.Short;
	END_IF


	bActionBusy	:= TRUE;

	fbOff(
		bError=> , 
		ipResultMessage=> , 
		bStart:= TRUE, 
		nAddress:= byAddr, 
		eAddressType:= eAddrType, 
		eCommandPriority:=Tc3_DALI.E_DALICommandPriority.Middle , 
		bBusy=> );
	
	IF NOT fbOff.bBusy	THEN
		IF	fbOff.bError	THEN
			bErr     	:= TRUE;
			nErrorId := fbOff.ipResultMessage.nEventId;

		END_IF
		bActionBusy		:= FALSE;
		fbOff(bStart:= FALSE);
	END_IF
END_ACTION

ACTION A_DALICmdQueryActualLevel:
	bActionBusy	:= TRUE;

	
fbQueryActualLevel(
	bError=> , 
	ipResultMessage=> , 
	bStart:= TRUE, 
	nAddress:= byShrtAdr, 
	eAddressType:= E_DALIAddressType.Short, 
	eCommandPriority:= E_DALICommandPriority.Middle, 
	bBusy=> , 
	nActualLevel=> );

	IF NOT fbQueryActualLevel.bBusy	THEN
		IF	fbQueryActualLevel.bError	THEN
			bErr     	:= TRUE;
			nErrorId := fbQueryActualLevel.ipResultMessage.nEventId;
		END_IF
		bActionBusy		:= FALSE;
		fbQueryActualLevel(bStart:= FALSE );
	END_IF
END_ACTION

ACTION A_DALICmdQueryMaxLevel:
	bActionBusy	:= TRUE;

fbQueryMaxLevel(
	bError=> , 
	ipResultMessage=> , 
	bStart:= TRUE, 
	nAddress:= byShrtAdr, 
	eAddressType:= E_DALIAddressType.Short, 
	eCommandPriority:= E_DALICommandPriority.Middle, 
	bBusy=> , 
	nMaxLevel=> );	
	


	IF NOT fbQueryMaxLevel.bBusy	THEN
		IF	fbQueryMaxLevel.bError	THEN
			bErr     	:= TRUE;
		END_IF
		bActionBusy		:= FALSE;
		fbQueryMaxLevel(bStart:= FALSE);
	END_IF
END_ACTION

ACTION A_DALICmdQueryMinLevel:
	bActionBusy	:= TRUE;

fbQueryMinLevel(
	bError=> , 
	ipResultMessage=> , 
	bStart:= TRUE, 
	nAddress:= byShrtAdr, 
	eAddressType:= E_DALIAddressType.Short, 
	eCommandPriority:= E_DALICommandPriority.Middle, 
	bBusy=> , 
	nMinLevel=> );	

	IF NOT fbQueryMinLevel.bBusy	THEN
		IF	fbQueryMinLevel.bError	THEN
			bErr     	:= TRUE;

		END_IF
		bActionBusy		:= FALSE;
		fbQueryMinLevel(bStart:= FALSE);
	END_IF
END_ACTION

ACTION A_DALICmdQueryPhysicalMinLevel:
	bActionBusy	:= TRUE;

	fbQueryPhysicalMinLevel(
		bError=> , 
		ipResultMessage=> , 
		bStart:= TRUE , 
		nAddress:= byShrtAdr, 
		eAddressType:= E_DALIAddressType.Short, 
		eCommandPriority:= E_DALICommandPriority.Middle, 
		bBusy=> , 
		nPhysicalMinimum=> );


	IF NOT fbQueryPhysicalMinLevel.bBusy	THEN
		IF	fbQueryPhysicalMinLevel.bError	THEN
			bErr     	:= TRUE;

		END_IF
		bActionBusy		:= FALSE;
		fbQueryPhysicalMinLevel(bStart:= FALSE);
	END_IF
END_ACTION

ACTION A_DALICmdRecallMaxLevel:
	IF emod = E_DALIAddressType.Group THEN
		byAddr		:= byGrpAdr;
		eAddrType	:= E_DALIAddressType.Group;
	ELSIF emod = E_DALIAddressType.Short THEN
		byAddr		:= byShrtAdr;
		eAddrType	:= E_DALIAddressType.Short;
	END_IF

	bActionBusy	:= TRUE;

	fbRecallMaxLevel(
		bError=> , 
		ipResultMessage=> , 
		bStart:= TRUE, 
		nAddress:= byAddr, 
		eAddressType:= eAddrType, 
		eCommandPriority:= E_DALICommandPriority.Middle, 
		bBusy=> );


	IF NOT fbRecallMaxLevel.bBusy	THEN
		IF	fbRecallMaxLevel.bError	THEN
			bErr     	:= TRUE;
		END_IF
		bActionBusy		:= FALSE;
		fbRecallMaxLevel(bStart:= FALSE);
	END_IF
END_ACTION

ACTION A_DALICmdRecallMinLevel:
	IF emod = E_DALIAddressType.Group THEN
		byAddr		:= byGrpAdr;
		eAddrType	:= E_DALIAddressType.Group;
	ELSIF emod = E_DALIAddressType.Short THEN
		byAddr		:= byShrtAdr;
		eAddrType	:= E_DALIAddressType.Short;
	END_IF


	bActionBusy	:= TRUE;

	fbRecallMinLevel(
		bError=> , 
		ipResultMessage=> , 
		bStart:= TRUE, 
		nAddress:= byAddr, 
		eAddressType:= eAddrType, 
		eCommandPriority:= E_DALICommandPriority.Middle, 
		bBusy=> );

	IF NOT fbRecallMinLevel.bBusy	THEN
		IF	fbRecallMinLevel.bError	THEN
			bErr     	:= TRUE;

		END_IF
		bActionBusy		:= FALSE;
		fbRecallMinLevel(bStart:= FALSE );
	END_IF
END_ACTION

ACTION A_DALICmdStepDown:
	IF emod = E_DALIAddressType.Group THEN
		byAddr		:= byGrpAdr;
		eAddrType	:= E_DALIAddressType.Group;
	ELSIF emod = E_DALIAddressType.Short THEN
		byAddr		:= byShrtAdr;
		eAddrType	:= E_DALIAddressType.Short;
	END_IF

	bActionBusy	:= TRUE;

	fbStepDown(
		bError=> , 
		ipResultMessage=> , 
		bStart:= TRUE, 
		nAddress:=byAddr , 
		eAddressType:= eAddrType, 
		eCommandPriority:= E_DALICommandPriority.Middle, 
		bBusy=> );


	IF NOT fbStepDown.bBusy	THEN
		IF	fbStepDown.bError	THEN
			bErr     	:= TRUE;
		END_IF
		bActionBusy		:= FALSE;
		fbStepDown(bStart:= FALSE );
	END_IF
END_ACTION

ACTION A_DALICmdStepUp:
	IF emod = E_DALIAddressType.Group THEN
		byAddr		:= byGrpAdr;
		eAddrType	:= E_DALIAddressType.Group;
	ELSIF emod = E_DALIAddressType.Short THEN
		byAddr		:= byShrtAdr;
		eAddrType	:= E_DALIAddressType.Short;
	END_IF


	bActionBusy	:= TRUE;

	fbStepUp(
		bError=> , 
		ipResultMessage=> , 
		bStart:= TRUE, 
		nAddress:=byAddr , 
		eAddressType:=eAddrType , 
		eCommandPriority:= E_DALICommandPriority.Middle, 
		bBusy=> );


	IF NOT fbStepUp.bBusy	THEN
		IF	fbStepUp.bError	THEN
			bErr     	:= TRUE;
			nErrorId := fbStepUp.ipResultMessage.nEventId;

		END_IF
		bActionBusy		:= FALSE;
		fbStepUp(bStart:= FALSE);
	END_IF
END_ACTION

ACTION A_DALICmdUp:
	IF emod = E_DALIAddressType.Group THEN
		byAddr		:= byGrpAdr;
		eAddrType	:= E_DALIAddressType.Group;
	ELSIF emod = E_DALIAddressType.Short THEN
		byAddr		:= byShrtAdr;
		eAddrType	:= E_DALIAddressType.Short;
	END_IF

	bActionBusy	:= TRUE;

	fbUp(
		bError=> , 
		ipResultMessage=> , 
		bStart:= TRUE , 
		nAddress:=byAddr , 
		eAddressType:= eAddrType, 
		eCommandPriority:= E_DALICommandPriority.High , 
		bBusy=> );

	IF NOT fbUp.bBusy	THEN
		IF	fbUp.bError	THEN
			bErr     	:= TRUE;
			nErrorId := fbUp.ipResultMessage.nEventId;
		END_IF
		bActionBusy		:= FALSE;
		fbUp(bStart:= FALSE );
	END_IF
END_ACTION

ACTION A_ResetRoutine:
	tonSeqTimer(IN:=FALSE);
	tonDimRepeat(IN:=FALSE);

	bErr     	:= FALSE;
	nErrorId 	:= 0;


	fbUp						(bStart:= FALSE );
	fbDwn						(bStart:= FALSE );
	fbOff						(bStart:= FALSE );
	fbRecallMaxLevel			(bStart:= FALSE );
	fbRecallMinLevel			(bStart:= FALSE );
	fbDirectArcPowerControl		(bStart:= FALSE );
	fbStepUp					(bStart:= FALSE );
	fbStepDown					(bStart:= FALSE );
	fbQueryActualLevel			(bStart:= FALSE );
	fbQueryPhysicalMinLevel		(bStart:= FALSE );
	fbQueryMinLevel				(bStart:= FALSE );
END_ACTION

{attribute 'monitoring' := 'call'}
PROPERTY ipDALICommunication : Tc3_DALI.I_DALICommunication
GET
ipDALICommunication := THIS^.ipCommunication;
END_GET
SET
THIS^.ipCommunicationPreset := ipDALICommunication;
END_SET
END_PROPERTY

//| Apply the perset value of IpCommunication if available
//| Return codes:
//|   FALSE: no peset value available
//|   TRUE: has taken the preset value
{attribute 'hide'}
METHOD PRIVATE TrySetCommunication : BOOL
VAR_INPUT
END_VAR
IF ((THIS^.ipCommunication <> THIS^.ipCommunicationPreset) AND (THIS^.ipCommunicationPreset <> 0)) THEN
	THIS^.ipCommunication := THIS^.ipCommunicationPreset;
	THIS^.fbUp.ipDALICommunication := THIS^.ipCommunication;
	THIS^.fbDwn.ipDALICommunication := THIS^.ipCommunication;
	THIS^.fbOff.ipDALICommunication := THIS^.ipCommunication;
	THIS^.fbRecallMaxLevel.ipDALICommunication := THIS^.ipCommunication;
	THIS^.fbRecallMinLevel.ipDALICommunication := THIS^.ipCommunication;
	THIS^.fbDirectArcPowerControl.ipDALICommunication := THIS^.ipCommunication;
	THIS^.fbStepUp.ipDALICommunication := THIS^.ipCommunication;	
	THIS^.fbStepDown.ipDALICommunication := THIS^.ipCommunication;
	THIS^.fbQueryActualLevel.ipDALICommunication := THIS^.ipCommunication;	
	THIS^.fbQueryMinLevel.ipDALICommunication := THIS^.ipCommunication;	
	THIS^.fbQueryMaxLevel.ipDALICommunication := THIS^.ipCommunication;
	THIS^.fbQueryPhysicalMinLevel.ipDALICommunication := THIS^.ipCommunication;
	THIS^.fbQueryActualLevelBackgound.ipDALICommunication := THIS^.ipCommunication;
	THIS^.fbQueryStatusBackground.ipDALICommunication := THIS^.ipCommunication;
	TrySetCommunication := TRUE;
ELSE
	TrySetCommunication := FALSE;
END_IF
END_METHOD

END_FUNCTION_BLOCK

// POUs/DALI/Ballast/FB_DALILgtCfg
FUNCTION_BLOCK FB_DALILgtCfg  (* V1.1 dfgdfgdfgdfgdfgfzxcv *)
VAR_INPUT
	byShrtAdr				: BYTE;
	byGrpAdr				: BYTE;
	eMod					: E_DALIAddressType:= E_DALIAddressType.Group;
	fMinCtrlVal			: REAL;
	fMaxCtrlVal			: REAL;
	eFadeTime				: E_DALIFadeTime:= E_DALIFadeTime.T02000ms;
	eFadeRate				: E_DALIFadeRate:= E_DALIFadeRate.N063StepsPerSec;
	uiBlinkTi				: UINT;
	uiOffDly				: UINT;
	bReInit					: BOOL;
	stLgtCmd				: ST_LgtCmd;
	DALI_LINE_NUM			: BYTE;
END_VAR
VAR_OUTPUT
	lrActlLgtLvl			: REAL;
	byActlLgtLvl			: BYTE;
	bLgt					: BOOL;
	lrActlMinCtrlVal		: REAL;
	bMinCtrlValRchd 		: BOOL;
	lrActlMaxCtrlVal		: REAL;
	bMaxCtrlValRchd 		: BOOL;
	lrRstVal				: REAL;
	eActlFadeTime			: E_DALIFadeTime;
	eActlFadeRate			: E_DALIFadeRate;
	byPhysMinVal			: BYTE;
	byActlMinCtrlVal		: BYTE;
	byActlMaxCtrlVal		: BYTE;
	bInitDevice				: BOOL;
	bBlinkSeqStarted 		: BOOL;
	bActionBusy				: BOOL;
	bErr     				: BOOL;
	nErrorId				: UDINT;
	byDALIDevSta			: BYTE;
END_VAR
VAR
	ipCommunication					: I_DALICommunication;
	ipCommunicationPreset			: I_DALICommunication;

	bInit					: BOOL;
	bBusy					: BOOL;
	bRstErr					: BOOL;
	rtReInit				: R_TRIG;
	bReactCmdSt				: BOOL;
	byAddr					: BYTE;
	eAddrType				: E_DALIAddressType;
	byArcPowerLevel			: BYTE;
	byDTR					: BYTE;
	uiCmdStep				: UINT;
	eFadeTime_SV			: E_DALIFadeTime;
	eFadeRate_SV			: E_DALIFadeRate;
	fMinCtrlVal_SV			: REAL;
	fMaxCtrlVal_SV			: REAL;
	bSetFadeRate			: BOOL;
	bSetFadeTime			: BOOL;
	bDimUp					: BOOL;
	bDimDwn					: BOOL;
	bySetFadeRate			: BYTE;
	bSetMinValInput			: BOOL;	(*Änderung MinVal über Bausteineingang*)
	bSetMaxValInput			: BOOL;	(*Änderung MaxVal über Bausteineingang*)
	bySetMinValInput		: BYTE;
	bySetMaxValInput		: BYTE;
	bSetMinValCmdSt			: BOOL;	(*Änderung MinVal über Kommandostruktur*)
	bSetMaxValCmdSt			: BOOL;	(*Änderung MaxVal über Kommandostruktur*)
	bySetMinValCmdSt		: BYTE;
	bySetMaxValCmdSt		: BYTE;
	byRstVal				: BYTE;
	bySttupCtrlVal			: BYTE;
	rtInitDevice			: R_TRIG;
	rtOff					: R_TRIG;
	rtClMinCtrlVal			: R_TRIG;
	rtClMaxCtrlVal			: R_TRIG;
	rtClOnVal				: R_TRIG;
	rtClRstVal				: R_TRIG;
	rtSetCtrlValDct			: R_TRIG;
	rtChgMaxCtrlVal			: R_TRIG;
	rtChgMinCtrlVal			: R_TRIG;
	rtStpUp							: R_TRIG;
	rtStpDwn						: R_TRIG;
	rtRmp							: R_TRIG;
	tonSeqTimer						: TON;
	tonDimRepeat					: TON;
	fbQueryActualLevel				: FB_DALI102QueryActualLevel(0);
	fbSetFadeRate					: FB_DALI102SetFadeRate(0);
	fbSetFadeTime					: FB_DALI102SetFadeTime(0);
	fbSetMinLevel					: FB_DALI102SetMinLevel(0);
	fbQueryMinLevel					: FB_DALI102QueryMinLevel(0);
	fbQueryMaxLevel					: FB_DALI102QueryMaxLevel(0);
	fbQueryPhysicalMinLevel			: FB_DALI102QueryPhysicalMinimum(0);
	fbSetMaxLevel					: FB_DALI102SetMaxLevel(0);
	fbSendValue						: FB_BA_ValTrigf;
	fbReTrigSend0					: R_TRIG;
	nStepQueryActualLevel			: UINT;
	tonCycleActualLevelMasterDev	: TON;
	bSetRetry						: BOOL;
	fbTimeOut						: TON;
	byActlFadeTime					: BYTE;

	nActualCount					: UDINT:= 1;
END_VAR
VAR_IN_OUT
END_VAR



{region "initialize the outputs"}
IF (NOT bInit) THEN
	THIS^.TrySetCommunication();		 
	bBusy := TRUE;
	nErrorId := 0;
	bErr := FALSE;
	bInit := TRUE;
END_IF
{endregion}


{region "check parameters"}
IF (ipCommunication = 0) THEN
	bErr := TRUE;
	nErrorId := TC_EVENTS.TcDALIEventClass.TheInterfaceToTheCommunicationBufferIsNotInitialized.nEventId;
	uiCmdStep := 0;
END_IF
IF ((eMod <> E_DALIAddressType.Short) AND (eMod <> E_DALIAddressType.Group) AND (eMod <> E_DALIAddressType.Broadcast) AND (eMod <> E_DALIAddressType.BroadcastUnaddr)) THEN
	bErr := TRUE;
	nErrorId := TC_EVENTS.TcDALIEventClass.ParameterAddressTypeLiesOutsideOfTheValidRange.nEventId;
	uiCmdStep := 0;
END_IF
IF ((eMod = E_DALIAddressType.Short) AND (byShrtAdr > 63)) THEN
	bErr := TRUE;
	nErrorId := TC_EVENTS.TcDALIEventClass.ParameterAddressIsAShortAddressAndLiesOutsideOfTheValidRange.nEventId;
	uiCmdStep := 0;
END_IF
IF ((eMod = E_DALIAddressType.Group) AND (byGrpAdr > 15)) THEN
	bErr := TRUE;
	nErrorId := TC_EVENTS.TcDALIEventClass.ParameterAddressIsAGroupAddressAndLiesOutsideOfTheValidRange.nEventId;
	uiCmdStep := 0;
END_IF
IF (byShrtAdr > 63) THEN
	bErr := TRUE;
	nErrorId := 16#8000; // custom error code: Parameter byShrtAdr lies outside of the valid range
	uiCmdStep := 0;
END_IF
	
IF (byGrpAdr > 15) THEN
	bErr := TRUE;
	nErrorId := 16#8001; // custom error code: Parameter byGrpAdr lies outside of the valid range
	uiCmdStep := 0;
END_IF
{endregion}

(*	bRstErr ist ein Fehlermerker: wenn vorher über Fehler, s.o. herausgesprungen wurde und nun "alles gut" ist,
dann hier Fehler einmalig zurücksetzen, damit im weiteren Verlauf die Warnmeldungen sichtbar werden können*)
IF	bRstErr  THEN
		bRstErr    	:= FALSE;
		bErr     	:= FALSE;
END_IF


(* + + + + + + + + + + + + + + + + + + + + + + + + + + + + + + + + + + + + + + + + + + + + *)
(*In den DALI-Ausführungsaktionen ist jedoch zur Sicherheit noch ein RETURN-Aussprung*)
IF (eMod=E_DALIAddressType.Short)	THEN
	bReactCmdSt:=FALSE;
ELSE
	bReactCmdSt:=TRUE;
END_IF

(* + + + + + + + + + + + + + + + + + + + + + + + + + + + + + + + + + + + + + + + + + + + + *)
(* + + + + + + + + + + + + + + + + + + + + + + + + + + + + + + + + + + + + + + + + + + + + *)
(*Init *)
rtReInit	 (CLK:=bReInit);
IF bReInit	THEN
	bInit:=FALSE;
END_IF

IF NOT bInit	THEN
	rtInitDevice		(CLK:=FALSE);
	bInitDevice			:= TRUE;
	fMinCtrlVal_SV		:= fMinCtrlVal;
	fMaxCtrlVal_SV		:= fMaxCtrlVal;
	bInit					:= TRUE;
END_IF

rtInitDevice (CLK:=bInitDevice);
bReactCmdSt:=TRUE;

(* + + + + + + + + + + + + + + + + + + + + + + + + + + + + + + + + + + + + + + + + + + + + *)
(*Change DimTime/FadeRate über Bausteineingang*)
IF	(eFadeTime<>eFadeTime_SV) OR rtInitDevice.Q THEN
	eFadeTime_SV	:= eFadeTime;
	IF NOT rtInitDevice.Q	THEN
		bSetFadeRate	:= TRUE;
	END_IF
END_IF

IF	(eFadeRate<>eFadeRate_SV) OR rtInitDevice.Q THEN
	eFadeRate_SV	:= eFadeRAte;
	IF NOT rtInitDevice.Q	THEN
		bSetFadeRate	:= TRUE;
	END_IF
END_IF

(* + + + + + + + + + + + + + + + + + + + + + + + + + + + + + + + + + + + + + + + + + + + + *)
(*Change Min-/MaxCtrlVal über Bausteineingang*)

IF	(fMinCtrlVal<>fMinCtrlVal_SV) OR rtInitDevice.Q THEN
	fMinCtrlVal_SV		:= fMinCtrlVal;
	IF 		fMinCtrlVal < 0.0		 THEN
		bySetMinValInput	:= 0;
	ELSIF	fMinCtrlVal > 100.0	 THEN
		bySetMinValInput	:= 254;
	ELSE
		bySetMinValInput := LIMIT(0,REAL_TO_BYTE(F_fDALICurve(fMinCtrlVal)), 254);
	END_IF
	IF NOT rtInitDevice.Q	THEN
		bSetMinValInput	:= TRUE;
	END_IF
END_IF

IF	(fMaxCtrlVal<>fMaxCtrlVal_SV) OR rtInitDevice.Q THEN
	fMaxCtrlVal_SV		:= fMaxCtrlVal;
	IF 		fMaxCtrlVal < 0.0		 THEN
		bySetMaxValInput	:= 0;
	ELSIF	fMaxCtrlVal > 100.0	 THEN
		bySetMaxValInput	:= 254;
	ELSE
		bySetMaxValInput := LIMIT(0,REAL_TO_BYTE(F_fDALICurve(fMaxCtrlVal)), 254);
	END_IF
	IF NOT rtInitDevice.Q	THEN
		bSetMaxValInput	:= TRUE;
	END_IF
END_IF


(* + + + + + + + + + + + + + + + + + + + + + + + + + + + + + + + + + + + + + + + + + + + + *)
(* Priorisierung aller Befehle und Schrittzuweisung *)
IF NOT bBusy	THEN
	IF			rtInitDevice.Q		THEN
				bBusy := TRUE;
				A_ResetRoutine();
				uiCmdStep:=1000;
	ELSIF		bSetFadeRate	 THEN
				bBusy := TRUE;
				A_ResetRoutine();
				uiCmdStep:=300;
	ELSIF	bSetMinValInput		 THEN
				bBusy := TRUE;
				A_ResetRoutine();
				uiCmdStep:=310;
	ELSIF	bSetMaxValInput		 THEN
				bBusy := TRUE;
				A_ResetRoutine();
				uiCmdStep:=320;
	ELSIF	bSetMinValCmdSt	 THEN
				bBusy := TRUE;
				A_ResetRoutine();
				uiCmdStep:=330;
	ELSIF	bSetMaxValCmdSt	 THEN
				bBusy := TRUE;
				A_ResetRoutine();
				uiCmdStep:=340;
	END_IF
END_IF

(* + + + + + + + + + + + + + + + + + + + + + + + + + + + + + + + + + + + + + + + + + + + + *)
(*Kommandoausgabe*)
CASE uiCmdStep OF

0: (*Idle*)
	bInitDevice := FALSE;
	bBusy := FALSE;

(* - - - - - - - - - - - - - - - - - - - - - - - - *)
300:(*Set new FadeRate*)
	bSetFadeRate:=FALSE;
	IF NOT bActionBusy	THEN
		IF bErr	THEN
			uiCmdStep:= 0;
		ELSE
			uiCmdStep:= 301;
		END_IF
	END_IF

301:(*Set new FadeRate*)
	A_DALICmdSetFadeRate();
	IF NOT bActionBusy	THEN
		uiCmdStep:= 0;
	END_IF
	eActlFadeRate:=eFadeRate;
	
	
305:(*Set new FadeTime *)
	bSetFadeTime:=FALSE;
	IF NOT bActionBusy	THEN
		IF bErr	THEN
			uiCmdStep:= 0;
		ELSE
			uiCmdStep:= 301;
		END_IF
	END_IF

306:(*Set new FadeRate*)
	A_DALICmdSetFadeRate();
	IF NOT bActionBusy	THEN
		uiCmdStep:= 0;
	END_IF
	eActlFadeTime:=eFadeTime;

(* - - - - - - - - - - - - - - - - - - - - - - - - *)
310:(*Set new Min-Level*)
	bSetMinValInput:=FALSE;

	byDTR:=bySetMinValInput;
	IF NOT bActionBusy	THEN
		IF bErr	THEN
			uiCmdStep:= 0;
		ELSE
			uiCmdStep:= 311;
		END_IF
	END_IF

311:(*Set new MinLevel*)
		A_DALICmdSetMinLevel_Input();
	IF NOT bActionBusy	THEN
		IF bErr	THEN
			uiCmdStep:= 0;
		ELSE
			uiCmdStep:= 350;
		END_IF
	END_IF

(* - - - - - - - - - - - - - - - - - - - - - - - - *)
320:(*Set new MaxLevel *)
	bSetMaxValInput:=FALSE;

	byDTR:=bySetMaxValInput;
	IF NOT bActionBusy	THEN
		IF bErr	THEN
			uiCmdStep:= 0;
		ELSE
			uiCmdStep:= 321;
		END_IF
	END_IF

321:(*Set new MaxLevel*)
		A_DALICmdSetMaxLevel_Input();
	IF NOT bActionBusy	THEN
		IF bErr	THEN
			uiCmdStep:= 0;
		ELSE
			uiCmdStep:= 350;
		END_IF
	END_IF

(* - - - - - - - - - - - - - - - - - - - - - - - - *)
330:(*Set new Min-Level *)
	bSetMinValCmdSt:=FALSE;

	byDTR:=bySetMinValCmdSt;
	IF NOT bActionBusy	THEN
		IF bErr	THEN
			uiCmdStep:= 0;
		ELSE
			uiCmdStep:= 331;
		END_IF
	END_IF

331:(*Set new MinLevel*)
		A_DALICmdSetMinLevel_CmdSt();
	IF NOT bActionBusy	THEN
		IF bErr	THEN
			uiCmdStep:= 0;
		ELSE
			uiCmdStep:= 350;
		END_IF
	END_IF

(* - - - - - - - - - - - - - - - - - - - - - - - - *)
340:(*Set new MaxLevel *)
	bSetMaxValCmdSt:=FALSE;

	byDTR:=bySetMaxValCmdSt;
	IF NOT bActionBusy	THEN
		IF bErr	THEN
			uiCmdStep:= 0;
		ELSE
			uiCmdStep:= 341;
		END_IF
	END_IF

341:(*Set new MaxLevel*)
		A_DALICmdSetMaxLevel_CmdSt();
	IF NOT bActionBusy	THEN
		IF bErr	THEN
			uiCmdStep:= 0;
		ELSE
			uiCmdStep:= 350;
		END_IF
	END_IF

(* - - - - - - - - - - - - - - - - - - - - - - - - *)
(*ZUR SICHERHEIT: ABFRAGE NACH PARAMETRIERUNG*)
350:(*Query Min Level*)
		A_DALICmdQueryMinLevel();
	IF NOT bActionBusy	THEN
		IF bErr	THEN
			uiCmdStep:= 0;
		ELSE
			uiCmdStep:= 351;
		END_IF
	END_IF
	byActlMinCtrlVal:=fbQueryMinLevel.nMinLevel;
	lrActlMinCtrlVal := LIMIT(0,REAL_TO_BYTE(F_fDALICurveRev(byActlMinCtrlVal)), 254);

351:(*Query Max Level*)
		A_DALICmdQueryMaxLevel();
	IF NOT bActionBusy	THEN
		IF bErr	THEN
			uiCmdStep:= 0;
		ELSE
			uiCmdStep:= 352;
		END_IF
	END_IF
	byActlMaxCtrlVal:=fbQueryMaxLevel.nMaxLevel;
	lrActlMaxCtrlVal := LIMIT(0,REAL_TO_BYTE(F_fDALICurveRev(byActlMaxCtrlVal)), 254);

352: (*Lichtabfrage wenn fertig*)
		A_DALICmdQueryActualLevel();
	IF NOT bActionBusy	THEN
		byActlLgtLvl	:= fbQueryActualLevel.nActualLevel;
		uiCmdStep		:= 0;
	END_IF

(* - - - - - - - - - - - - - - - - - - - - - - - - *)
(*Init Device-Routine*)

1000: (*Wait fort free DT8*)
	IF NOT arrbBlockDTR[DALI_LINE_NUM] THEN
		uiCmdStep:= 1001;
		arrbBlockDTR[DALI_LINE_NUM]:= TRUE;
		bActionBusy:= FALSE;
	END_IF

1001:(*Set new FadeRate *)
		IF NOT bActionBusy	THEN
			IF bErr	THEN
				uiCmdStep:= 0;
				arrbBlockDTR[DALI_LINE_NUM]:=FALSE;
			ELSE
				uiCmdStep:= 1002;
			END_IF
		END_IF

1002:(*Set new FadeRate*)
	A_DALICmdSetFadeRate();
	IF NOT bActionBusy	THEN
		IF bErr	THEN
			uiCmdStep:= 0;
			arrbBlockDTR[DALI_LINE_NUM]:=FALSE;
		ELSE
			uiCmdStep:= 1003;
		END_IF
	END_IF
	eActlFadeRate:=eFadeRate;

1003:(*Set new FadeTime*)
	eFadeTime_SV:= DALI_Param.eGlobalFadeTime;
	A_DALICmdSetFadeTime();
	IF NOT bActionBusy	THEN
		IF bErr	THEN
			uiCmdStep:= 0;
			arrbBlockDTR[DALI_LINE_NUM]:=FALSE;
		ELSE
			uiCmdStep:= 1005;
		END_IF
	END_IF
	eActlFadeTime:=eFadeTime_SV;
	
1005:(*Set new FadeTime *)
	eFadeTime_SV:=eGlobalFadeTime;
	IF NOT bActionBusy	THEN
		IF bErr	THEN
			uiCmdStep:= 0;
			arrbBlockDTR[DALI_LINE_NUM]:=FALSE;
		ELSE
			uiCmdStep:= 1006;
		END_IF
	END_IF

1006:(*Set new FadeTime*)
	A_DALICmdSetFadeTime();
	IF NOT bActionBusy	THEN
		IF bErr	THEN
			uiCmdStep:= 0;
			arrbBlockDTR[DALI_LINE_NUM]:=FALSE;
		ELSE
			uiCmdStep:= 1010;
		END_IF
	END_IF
	byActlFadeTime:=eFadeTime_SV;


1010:(*Set new Min-Level *)
	byDTR:=bySetMinValInput;
	IF NOT bActionBusy	THEN
		IF bErr	THEN
			uiCmdStep:= 0;
			arrbBlockDTR[DALI_LINE_NUM]:=FALSE;
		ELSE
			uiCmdStep:= 1015;
		END_IF
	END_IF

1015:(*Set new Min-Level*)
		A_DALICmdSetMinLevel_Input();
	IF NOT bActionBusy	THEN
		IF bErr	THEN
			uiCmdStep:= 0;
			arrbBlockDTR[DALI_LINE_NUM]:=FALSE;
		ELSE
			uiCmdStep:= 1020;
		END_IF
	END_IF

1020:(*Set new MaxLevel*)
	byDTR:=bySetMaxValInput;
	IF NOT bActionBusy	THEN
		IF bErr	THEN
			uiCmdStep:= 0;
			arrbBlockDTR[DALI_LINE_NUM]:=FALSE;
		ELSE
			uiCmdStep:= 1025;
		END_IF
	END_IF

1025:(*Set new MaxLevel*)
		A_DALICmdSetMaxLevel_Input();
	IF NOT bActionBusy	THEN
		IF bErr	THEN
			uiCmdStep:= 0;
			arrbBlockDTR[DALI_LINE_NUM]:=FALSE;
		ELSE
			uiCmdStep:= 1030;
		END_IF
	END_IF

1030:(*Query physical Min Level*)
		A_DALICmdQueryPhysicalMinLevel();
	IF NOT bActionBusy	THEN
		IF bErr	THEN
			uiCmdStep:= 0;
			arrbBlockDTR[DALI_LINE_NUM]:=FALSE;
		ELSE
			uiCmdStep:= 1035;
		END_IF
	END_IF
	byPhysMinVal:=fbQueryPhysicalMinLevel.nPhysicalMinimum;

1035:(*Query Min Level*)
		A_DALICmdQueryMinLevel();
	IF NOT bActionBusy	THEN
		IF bErr	THEN
			uiCmdStep:= 0;
			arrbBlockDTR[DALI_LINE_NUM]:=FALSE;
		ELSE
			uiCmdStep:= 1040;
		END_IF
	END_IF
	byActlMinCtrlVal:=fbQueryMinLevel.nMinLevel;
	lrActlMinCtrlVal := LIMIT(0,REAL_TO_BYTE(F_fDALICurveRev(byActlMinCtrlVal)), 254);

1040:(*Query Max Level*)
		A_DALICmdQueryMaxLevel();
	IF NOT bActionBusy	THEN
		IF bErr	THEN
			uiCmdStep:= 0;
			arrbBlockDTR[DALI_LINE_NUM]:=FALSE;
		ELSE
			uiCmdStep:= 1050;
		END_IF
	END_IF
	byActlMaxCtrlVal:=fbQueryMaxLevel.nMaxLevel;
	lrActlMaxCtrlVal := LIMIT(0,REAL_TO_BYTE(F_fDALICurveRev(byActlMaxCtrlVal)), 254);

1050: (*Lichtabfrage wenn fertig*)
		A_DALICmdQueryActualLevel();
	IF NOT bActionBusy	THEN
		byActlLgtLvl	:= fbQueryActualLevel.nActualLevel;
		uiCmdStep		:= 0;
		arrbBlockDTR[DALI_LINE_NUM]:=FALSE;
	END_IF

END_CASE
	
(* + + + + + + + + + + + + + + + + + + + + + + + + + + + + + + + + + + + + + + + + + + + + *)
(*Umrechnung des Lichtwertes lrActlLgtLvl und Speicherung des letzten Wertes vor Aus*)

bMinCtrlValRchd:=(byActlLgtLvl=byActlMinCtrlVal);
bMaxCtrlValRchd:=(byActlLgtLvl=byActlMaxCtrlVal);

ACTION A_DALICmdQueryActualLevel:
	bActionBusy	:= TRUE;

	
fbQueryActualLevel(
	bError=> , 
	ipResultMessage=> , 
	bStart:= TRUE, 
	nAddress:= byShrtAdr, 
	eAddressType:= E_DALIAddressType.Short, 
	eCommandPriority:= E_DALICommandPriority.Middle, 
	bBusy=> , 
	nActualLevel=> );

	IF NOT fbQueryActualLevel.bBusy	THEN
		IF	fbQueryActualLevel.bError	THEN
			bErr     	:= TRUE;
			nErrorId := fbQueryActualLevel.ipResultMessage.nEventId;
		END_IF
		bActionBusy		:= FALSE;
		fbQueryActualLevel(bStart:= FALSE );
	END_IF
END_ACTION

ACTION A_DALICmdQueryMaxLevel:
	bActionBusy	:= TRUE;

fbQueryMaxLevel(
	bError=> , 
	ipResultMessage=> , 
	bStart:= TRUE, 
	nAddress:= byShrtAdr, 
	eAddressType:= E_DALIAddressType.Short, 
	eCommandPriority:= E_DALICommandPriority.Middle, 
	bBusy=> , 
	nMaxLevel=> );	
	


	IF NOT fbQueryMaxLevel.bBusy	THEN
		IF	fbQueryMaxLevel.bError	THEN
			bErr     	:= TRUE;
		END_IF
		bActionBusy		:= FALSE;
		fbQueryMaxLevel(bStart:= FALSE);
	END_IF
END_ACTION

ACTION A_DALICmdQueryMinLevel:
	bActionBusy	:= TRUE;

fbQueryMinLevel(
	bError=> , 
	ipResultMessage=> , 
	bStart:= TRUE, 
	nAddress:= byShrtAdr, 
	eAddressType:= E_DALIAddressType.Short, 
	eCommandPriority:= E_DALICommandPriority.Middle, 
	bBusy=> , 
	nMinLevel=> );	

	IF NOT fbQueryMinLevel.bBusy	THEN
		IF	fbQueryMinLevel.bError	THEN
			bErr     	:= TRUE;

		END_IF
		bActionBusy		:= FALSE;
		fbQueryMinLevel(bStart:= FALSE);
	END_IF
END_ACTION

ACTION A_DALICmdQueryPhysicalMinLevel:
	bActionBusy	:= TRUE;

	fbQueryPhysicalMinLevel(
		bError=> , 
		ipResultMessage=> , 
		bStart:= TRUE , 
		nAddress:= byShrtAdr, 
		eAddressType:= E_DALIAddressType.Short, 
		eCommandPriority:= E_DALICommandPriority.Middle, 
		bBusy=> , 
		nPhysicalMinimum=> );


	IF NOT fbQueryPhysicalMinLevel.bBusy	THEN
		IF	fbQueryPhysicalMinLevel.bError	THEN
			bErr     	:= TRUE;

		END_IF
		bActionBusy		:= FALSE;
		fbQueryPhysicalMinLevel(bStart:= FALSE);
	END_IF
END_ACTION

ACTION A_DALICmdSetFadeRate:
	IF emod = E_DALIAddressType.Group THEN
		byAddr		:= byGrpAdr;
		eAddrType	:= E_DALIAddressType.Group;
	ELSIF emod = E_DALIAddressType.Short THEN
		byAddr		:= byShrtAdr;
		eAddrType	:= E_DALIAddressType.Short;
	END_IF

	bActionBusy	:= TRUE;

	fbSetFadeRate(
		bError=> , 
		ipResultMessage=> , 
		bStart:= TRUE, 
		nAddress:= byAddr , 
		eAddressType:= eAddrType , 
		eCommandPriority:=Tc3_DALI.E_DALICommandPriority.Middle , 
		bBusy=> , 
		eFadeRate:=eFadeRate );
	
	IF (NOT fbSetFadeRate.bBusy) THEN
		IF fbSetFadeRate.bError THEN
			bErr := TRUE;
			nErrorId := fbSetFadeRate.ipResultMessage.nEventId;
		END_IF
		bActionBusy		:= FALSE;
		fbSetFadeRate(bStart:= FALSE);
	END_IF
END_ACTION

ACTION A_DALICmdSetFadeTime:
	IF emod = E_DALIAddressType.Group THEN
		byAddr		:= byGrpAdr;
		eAddrType	:= E_DALIAddressType.Group;
	ELSIF emod = E_DALIAddressType.Short THEN
		byAddr		:= byShrtAdr;
		eAddrType	:= E_DALIAddressType.Short;
	END_IF


	bActionBusy	:= TRUE;

	fbSetFadeTime(
		bError=> , 
		ipResultMessage=> , 
		bStart:= TRUE, 
		nAddress:= byAddr , 
		eAddressType:= eAddrType , 
		eCommandPriority:=Tc3_DALI.E_DALICommandPriority.Middle , 
		bBusy=> , 
		eFadeTime:=eFadeTime_SV );
	
	IF (NOT fbSetFadeTime.bBusy) THEN
		IF fbSetFadeTime.bError THEN
			bErr := TRUE;
			nErrorId := fbSetFadeTime.ipResultMessage.nEventId;
		END_IF
		bActionBusy		:= FALSE;
		fbSetFadeTime(bStart:= FALSE);
	END_IF
END_ACTION

ACTION A_DALICmdSetMaxLevel_CmdSt:


	IF emod = E_DALIAddressType.Group THEN
		byAddr		:= byGrpAdr;
		eAddrType	:= E_DALIAddressType.Group;
	ELSIF emod = E_DALIAddressType.Short THEN
		byAddr		:= byShrtAdr;
		eAddrType	:= E_DALIAddressType.Short;
	END_IF


	bActionBusy	:= TRUE;

	fbSetMaxLevel(
		bError=> , 
		ipResultMessage=> , 
		bStart:= TRUE, 
		nAddress:= byAddr , 
		eAddressType:= eAddrType , 
		eCommandPriority:=Tc3_DALI.E_DALICommandPriority.Middle , 
		bBusy=> , 
		nMaxLevel:= byDTR);
	

	IF (NOT fbSetMaxLevel.bBusy) THEN
		IF fbSetMaxLevel.bError THEN
			bErr := TRUE;
			nErrorId := fbSetMaxLevel.ipResultMessage.nEventId;
		END_IF
		bActionBusy		:= FALSE;
		fbSetMaxLevel(bStart:= FALSE);
	END_IF
END_ACTION

ACTION A_DALICmdSetMaxLevel_Input:


	IF emod = E_DALIAddressType.Group THEN
		byAddr		:= byGrpAdr;
		eAddrType	:= E_DALIAddressType.Group;
	ELSIF emod = E_DALIAddressType.Short THEN
		byAddr		:= byShrtAdr;
		eAddrType	:= E_DALIAddressType.Short;
	END_IF


	bActionBusy	:= TRUE;

	fbSetMaxLevel(
		bError=> , 
		ipResultMessage=> , 
		bStart:= TRUE, 
		nAddress:= byAddr , 
		eAddressType:= eAddrType , 
		eCommandPriority:=Tc3_DALI.E_DALICommandPriority.Middle , 
		bBusy=> , 
		nMaxLevel:= byDTR);
	

	IF (NOT fbSetMaxLevel.bBusy) THEN
		IF fbSetMaxLevel.bError THEN
			bErr := TRUE;
			nErrorId := fbSetMaxLevel.ipResultMessage.nEventId;
		END_IF
		bActionBusy		:= FALSE;
		fbSetMaxLevel(bStart:= FALSE);
	END_IF
END_ACTION

ACTION A_DALICmdSetMinLevel_CmdSt:

	IF emod = E_DALIAddressType.Group THEN
		byAddr		:= byGrpAdr;
		eAddrType	:= E_DALIAddressType.Group;
	ELSIF emod = E_DALIAddressType.Short THEN
		byAddr		:= byShrtAdr;
		eAddrType	:= E_DALIAddressType.Short;
	END_IF


	bActionBusy	:= TRUE;

	fbSetMinLevel(
		bError=> , 
		ipResultMessage=> , 
		bStart:= TRUE, 
		nAddress:= byAddr , 
		eAddressType:= eAddrType , 
		eCommandPriority:=Tc3_DALI.E_DALICommandPriority.Middle , 
		bBusy=> , 
		nMinLevel:= byDTR);
	

	IF (NOT fbSetMinLevel.bBusy) THEN
		IF fbSetMinLevel.bError THEN
			bErr := TRUE;
			nErrorId := fbSetMinLevel.ipResultMessage.nEventId;
		END_IF
		bActionBusy		:= FALSE;
		fbSetMinLevel(bStart:= FALSE);
	END_IF
END_ACTION

ACTION A_DALICmdSetMinLevel_Input:
	IF emod = E_DALIAddressType.Group THEN
		byAddr		:= byGrpAdr;
		eAddrType	:= E_DALIAddressType.Group;
	ELSIF emod = E_DALIAddressType.Short THEN
		byAddr		:= byShrtAdr;
		eAddrType	:= E_DALIAddressType.Short;
	END_IF


	bActionBusy	:= TRUE;

	fbSetMinLevel(
		bError=> , 
		ipResultMessage=> , 
		bStart:= TRUE, 
		nAddress:= byAddr , 
		eAddressType:= eAddrType , 
		eCommandPriority:=Tc3_DALI.E_DALICommandPriority.Middle , 
		bBusy=> , 
		nMinLevel:= byDTR);
	

	IF (NOT fbSetMinLevel.bBusy) THEN
		IF fbSetMinLevel.bError THEN
			bErr := TRUE;
			nErrorId := fbSetMinLevel.ipResultMessage.nEventId;
		END_IF
		bActionBusy		:= FALSE;
		fbSetMinLevel(bStart:= FALSE);
	END_IF
END_ACTION

ACTION A_ResetRoutine:
	tonSeqTimer(IN:=FALSE);
	tonDimRepeat(IN:=FALSE);

	bErr     	:= FALSE;
	nErrorId 	:= 0;

	fbQueryActualLevel			(bStart:= FALSE );
	fbSetFadeRate				(bStart:= FALSE );
	fbSetFadeTime				(bStart:= FALSE );
	fbQueryPhysicalMinLevel		(bStart:= FALSE );
	fbSetMinLevel				(bStart:= FALSE );
	fbQueryMinLevel				(bStart:= FALSE );
	fbSetMaxLevel				(bStart:= FALSE );
END_ACTION

{attribute 'monitoring' := 'call'}
PROPERTY ipDALICommunication : Tc3_DALI.I_DALICommunication
GET
ipDALICommunication := THIS^.ipCommunication;
END_GET
SET
THIS^.ipCommunicationPreset := ipDALICommunication;
END_SET
END_PROPERTY

//| Apply the perset value of IpCommunication if available
//| Return codes:
//|   FALSE: no peset value available
//|   TRUE: has taken the preset value
{attribute 'hide'}
METHOD PRIVATE TrySetCommunication : BOOL
VAR_INPUT
END_VAR
IF ((THIS^.ipCommunication <> THIS^.ipCommunicationPreset) AND (THIS^.ipCommunicationPreset <> 0)) THEN
	THIS^.ipCommunication := THIS^.ipCommunicationPreset;

	THIS^.fbQueryActualLevel.ipDALICommunication := THIS^.ipCommunication;	
	THIS^.fbSetFadeRate.ipDALICommunication := THIS^.ipCommunication;
	THIS^.fbSetFadeTime.ipDALICommunication := THIS^.ipCommunication;
	THIS^.fbSetMaxLevel.ipDALICommunication := THIS^.ipCommunication;
	THIS^.fbSetMinLevel.ipDALICommunication := THIS^.ipCommunication;
	THIS^.fbQueryMinLevel.ipDALICommunication := THIS^.ipCommunication;	
	THIS^.fbQueryMaxLevel.ipDALICommunication := THIS^.ipCommunication;
	THIS^.fbQueryPhysicalMinLevel.ipDALICommunication := THIS^.ipCommunication;
	TrySetCommunication := TRUE;
ELSE
	TrySetCommunication := FALSE;
END_IF
END_METHOD

END_FUNCTION_BLOCK

// POUs/DALI/Ballast/FB_Light_Ballast
FUNCTION_BLOCK FB_Light_Ballast 
VAR_OUTPUT
	bLgt_Prim							: BOOL;	(*Light is either on or off*)
	fActlLgtLvl_Prim					: REAL;(*Actual light-level in %*)
	byActlLgtLvl_Prim					: BYTE;	(*Actual light-level in 0..254*)
	bError_Prim 						: BOOL;
	nError_Prim 						: UINT;	
	bLgt_Sec							: BOOL;	(*Light is either on or off*)
	fActlLgtLvl_Sec						: REAL;(*Actual light-level in %*)
	byActlLgtLvl_Sec					: BYTE;	(*Actual light-level in 0..254*)
	
	bLgt_Supl							: BOOL;	(*Light is either on or off*)
	fActlLgtLvl_Supl					: REAL;(*Actual light-level in %*)
	byActlLgtLvl_Supl					: BYTE;	(*Actual light-level in 0..254*)
END_VAR
VAR_INPUT CONSTANT
	nCycleTimeInMS						: UDINT;
END_VAR
VAR

//Global settings for both groups

	eFadeTime							: E_DALIFadeTime:= E_DALIFadeTime.T02000ms;	
	eFadeRate							: E_DALIFadeRate:= E_DALIFadeRate.N063StepsPerSec;		

//Primary group of lamps
	fbLgtActr_Prim						: FB_DALILgtActr_EX;		
// Input parameter for Prim row							

	fPrim_MinCtrlVal					: REAL := 0;	(*Minimum light-value in %*)				
	fPrim_MaxCtrlVal					: REAL := 100;	(*Maximum light-value in %*)				
	fPrim_LgtOffset						: REAL := 0;	(*Light-offset-value in %*)				
	nPrim_BlinkTi						: UINT := 0;	(*Blinking-sequence Off-pulse in s*)			
	nPrim_OffDly						: UINT := 0;	(*Blinking-sequence On-Time after Off-pulse in s*)			
	nPrim_PollActLgtLvl					: UINT := 30;	(*Polling-interval light-value/statusbyte*)					
	bPrim_ReInit						: BOOL;			(*Restart Init-Routine*)	
// Status variables for Primdow row							
	fPrim_ActlMinCtrlVal				: REAL;	(*Currently programmed min-value in %*)			
	bPrim_MinCtrlValRchd				: BOOL;	(*Min-value reached*)			
	fPrim_ActlMaxCtrlVal				: REAL;	(*Currently programmed max-value in %*)			
	bPrim_MaxCtrlValRchd				: BOOL;	(*Max-value reached*)			
	fPrim_RstVal						: REAL;	(*Actual reset-value in %*)			
	ePrim_ActlFadeTime					: E_DALIFadeTime;	(*Currently programmed fade-rate*)			
	ePrim_ActlFadeRate					: E_DALIFadeRate;	(*Currently programmed fade-rate*)			
	nPrim_PhysMinVal					: BYTE;	(*phys. Min-Value in 0..254*)			
	nPrim_ActlMinCtrlVal				: BYTE;	(*Currently programmed min-value in 0..254*)			
	nPrim_ActlMaxCtrlVal				: BYTE;	(*Currently programmed max-value in 0..254*)			
	bPrim_InitDevice					: BOOL;	(*Init-routine*)			
	bPrim_BlinkSeqStarted				: BOOL;	(*Blinking-sequence started*)			
	bPrim_ActionBusy					: BOOL;	(*DALI-command is being executed*)			
	bPrim_Err							: BOOL;	(*Module in error-state*)			
	nPrim_ErrId							: UDINT;	(*ErrorId*)			
	nPrim_DALIDevSta					: BYTE;	(*DALI-Statusbyte*)			
	fbMasterSelectorPrim				: FB_MasterSelector;

//Secondary Row
	fbLgtActr_Sec						: FB_DALILgtActr_EX;		
// Input parameter for Sec row							
	fSec_MinCtrlVal						: REAL := 0;	(*Minimum light-value in %*)					
	fSec_MaxCtrlVal						: REAL := 100;	(*Maximum light-value in %*)					
	fSec_LgtOffset						: REAL := 0;	(*Light-offset-value in %*)				
	nSec_BlinkTi						: UINT := 0;	(*Blinking-sequence Off-pulse in s*)				
	nSec_OffDly							: UINT := 0;	(*Blinking-sequence On-Time after Off-pulse in s*)				
	nSec_PollActLgtLvl					: UINT := 30;	(*Polling-interval light-value/statusbyte*)					
	bSec_ReInit							: BOOL;			(*Restart Init-Routine*)		
// Status variables for Secdow row												
	fSec_ActlMinCtrlVal					: REAL;	(*Currently programmed min-value in %*)						
	bSec_MinCtrlValRchd					: BOOL;	(*Min-value reached*)						
	fSec_ActlMaxCtrlVal				: REAL;	(*Currently programmed max-value in %*)						
	bSec_MaxCtrlValRchd					: BOOL;	(*Max-value reached*)						
	fSec_RstVal							: REAL;	(*Actual reset-value in %*)				
	eSec_ActlFadeTime					: E_DALIFadeTime;	(*Currently programmed fade-rate*)					
	eSec_ActlFadeRate					: E_DALIFadeRate;	(*Currently programmed fade-rate*)					
	nSec_PhysMinVal						: BYTE;	(*phys. Min-Value in 0..254*)					
	nSec_ActlMinCtrlVal					: BYTE;	(*Currently programmed min-value in 0..254*)						
	nSec_ActlMaxCtrlVal					: BYTE;	(*Currently programmed max-value in 0..254*)						
	bSec_InitDevice						: BOOL;	(*Init-routine*)					
	bSec_BlinkSeqStarted				: BOOL;	(*Blinking-sequence started*)						
	bSec_ActionBusy						: BOOL;	(*DALI-command is being executed*)					
	bSec_Err							: BOOL;	(*Module in error-state*)			
	nSec_ErrId							: UDINT;	(*ErrorId*)			
	nSec_DALIDevSta						: BYTE;	(*DALI-Statusbyte*)					
	
	fbMasterSelectorSec					: FB_MasterSelector;

	fbLgtActr_Supl						: FB_DALILgtActr_EX;			
// Input parameter for Supl row										
	fSupl_MinCtrlVal						: REAL := 0;	(*Minimum light-value in %*)					
	fSupl_MaxCtrlVal						: REAL := 100;	(*Maximum light-value in %*)					
	fSupl_LgtOffset						: REAL := 0;	(*Light-offset-value in %*)					
	nSupl_BlinkTi						: UINT := 0;	(*Blinking-sequence Off-pulse in s*)					
	nSupl_OffDly							: UINT := 0;	(*Blinking-sequence On-Time after Off-pulse in s*)				
	nSupl_PollActLgtLvl					: UINT := 30;	(*Polling-interval light-value/statusbyte*)						
	bSupl_ReInit							: BOOL;			(*Restart Init-Routine*)		
// Status variables for Supldow row													
	fSupl_ActlMinCtrlVal					: REAL;	(*Currently programmed min-value in %*)						
	bSupl_MinCtrlValRchd					: BOOL;	(*Min-value reached*)						
	fSupl_ActlMaxCtrlVal				: REAL;	(*Currently programmed max-value in %*)							
	bSupl_MaxCtrlValRchd					: BOOL;	(*Max-value reached*)						
	fSupl_RstVal							: REAL;	(*Actual reset-value in %*)				
	eSupl_ActlFadeTime					: E_DALIFadeTime;	(*Currently programmed fade-rate*)						
	eSupl_ActlFadeRate					: E_DALIFadeRate;	(*Currently programmed fade-rate*)						
	nSupl_PhysMinVal						: BYTE;	(*phys. Min-Value in 0..254*)					
	nSupl_ActlMinCtrlVal					: BYTE;	(*Currently programmed min-value in 0..254*)						
	nSupl_ActlMaxCtrlVal					: BYTE;	(*Currently programmed max-value in 0..254*)						
	bSupl_InitDevice						: BOOL;	(*Init-routine*)					
	bSupl_BlinkSeqStarted				: BOOL;	(*Blinking-sequence started*)							
	bSupl_ActionBusy						: BOOL;	(*DALI-command is being executed*)					
	bSupl_Err							: BOOL;	(*Module in error-state*)				
	nSupl_ErrId							: UDINT;	(*ErrorId*)				
	nSupl_DALIDevSta						: BYTE;	(*DALI-Statusbyte*)					
			
	fbMasterSelectorSupl				: FB_MasterSelector;					
	
END_VAR

METHOD M_PrimBallast : BOOL
VAR_INPUT
	byShrtAdr_Prim						: BYTE:=1;	
	byGrpAdr_Prim						: BYTE := 3;	
	eMod_Prim							: E_DALIAddressType := E_DALIADDRESSTYPE.Group;
	stLgtCmd_Prim						: ST_LgtCmd;	(*Kommandostruktur // command-structure*)
	DALI_LINE_NUM						: BYTE ;	(*DALI-Linie//DALI-line*)
	bUseGlobalFadeTimeSettings			: BOOL := TRUE;
	bReInit								: BOOL;	(*Restart Init-Routine*)
	bTurnOff							: BOOL;	(*Start ramp to 0%*)	
	ipCommunication						: Tc3_DALI.I_DALICommunication;
END_VAR

VAR
END_VAR

fbLgtActr_Prim.ipDALICommunication:= ipCommunication;

IF (ipCommunication <> 0) AND (DALI_LINE_NUM <> 0) THEN

	IF eMod_Prim = E_DALIAddressType.Group THEN
		IF g_arrDiagnosisRunOnce[DALI_LINE_NUM] THEN
			fbMasterSelectorPrim(
				bErrFromBallastFB:=fbLgtActr_Prim.bErr , 
				byGrpAdr:= byGrpAdr_Prim, 
				DALI_LINE_NUM:= DALI_LINE_NUM, 
				nMasterUnitID=> byShrtAdr_Prim, 
				stGroupSorter:= GVL_DALI.g_arrAddrInGroups[DALI_LINE_NUM]);
		END_IF		
	END_IF
	

(* For checking which task the FB are called*)
	IF g_arrDiagnosisRunOnce[DALI_LINE_NUM] THEN
		fbLgtActr_Prim(	
			byShrtAdr:= byShrtAdr_Prim, 
			byGrpAdr:= byGrpAdr_Prim, 
			eMod:= eMod_Prim, 
			fSttupCtrlVal:= stLgtCmd_Prim.fSetCtrlValDct, 
			fMinCtrlVal:= fPrim_MinCtrlVal, 
			fMaxCtrlVal:= fPrim_MaxCtrlVal, 
			fLgtOffset:= fPrim_LgtOffset, 
			eFadeTime:= SEL(bUseGlobalFadeTimeSettings, eFadeTime, eGlobalFadeTime), 
			eFadeRate:= eFadeRate, 
			uiBlinkTi:= nPrim_BlinkTi, 
			uiOffDly:= nPrim_OffDly, 
			uiPollActLgtLvl:= nPrim_PollActLgtLvl, 
			bReInit:= bPrim_ReInit, 
			nCycleTimeInMS:= nCycleTimeInMS,
			stLgtCmd:= stLgtCmd_Prim, 
			DALI_LINE_NUM:= DALI_LINE_NUM, 
			fActlLgtLvl=> fActlLgtLvl_Prim, 
			byActlLgtLvl=> byActlLgtLvl_Prim, 
			bLgt=> bLgt_Prim, 
			fActlMinCtrlVal=> fPrim_ActlMinCtrlVal, 
			bMinCtrlValRchd=> bPrim_MinCtrlValRchd, 
			fActlMaxCtrlVal=> fPrim_ActlMaxCtrlVal, 
			bMaxCtrlValRchd=> bPrim_MaxCtrlValRchd, 
			fRstVal=>fPrim_RstVal, 
			eActlFadeTime=> ePrim_ActlFadeTime, 
			eActlFadeRate=> ePrim_ActlFadeRate, 
			byPhysMinVal=> nPrim_PhysMinVal, 
			byActlMinCtrlVal=> nPrim_ActlMinCtrlVal, 
			byActlMaxCtrlVal=> nPrim_ActlMaxCtrlVal, 
			bInitDevice=> bPrim_InitDevice, 
			bBlinkSeqStarted=> bPrim_BlinkSeqStarted, 
			bActionBusy=> bPrim_ActionBusy, 
			bErr=> bPrim_Err, 
			nErrorId=> nPrim_ErrId, 
			byDALIDevSta=> nPrim_DALIDevSta);
	END_IF

END_IF
END_METHOD

METHOD M_SecBallast : BOOL
VAR_INPUT
	byShrtAdr_Sec						: BYTE:=3;	
	byGrpAdr_Sec						: BYTE := 4	;
	eMod_Sec							: E_DALIAddressType := E_DALIADDRESSTYPE.Group;
	stLgtCmd_Sec						: ST_LgtCmd;	(*Kommandostruktur // command-structure*)
	DALI_LINE_NUM						: BYTE ;	(*DALI-Linie//DALI-line*)
	bUseGlobalFadeTimeSettings			: BOOL := TRUE;
	bReInit								: BOOL;	(*Restart Init-Routine*)
	bTurnOff							: BOOL;	(*Start ramp to 0%*)	
	ipCommunication						: Tc3_DALI.I_DALICommunication;
END_VAR


fbLgtActr_Sec.ipDALICommunication:= ipCommunication;

IF (ipCommunication <> 0) AND (DALI_LINE_NUM <> 0) THEN

	IF eMod_Sec = E_DALIAddressType.Group THEN
		IF g_arrDiagnosisRunOnce[DALI_LINE_NUM] THEN
			fbMasterSelectorSec(
				bErrFromBallastFB:=fbLgtActr_Sec.bErr , 
				byGrpAdr:= byGrpAdr_Sec, 
				DALI_LINE_NUM:= DALI_LINE_NUM, 
				nMasterUnitID=> byShrtAdr_Sec, 
				stGroupSorter:= GVL_DALI.g_arrAddrInGroups[DALI_LINE_NUM]);
		END_IF
	END_IF

	IF g_arrDiagnosisRunOnce[DALI_LINE_NUM] THEN	
		fbLgtActr_Sec(	
			byShrtAdr:= byShrtAdr_Sec, 
			byGrpAdr:= byGrpAdr_Sec, 
			eMod:= eMod_Sec, 
			fSttupCtrlVal:= stLgtCmd_Sec.fSetCtrlValDct, 
			fMinCtrlVal:= fSec_MinCtrlVal, 
			fMaxCtrlVal:= fSec_MaxCtrlVal, 
			fLgtOffset:= fSec_LgtOffset, 
			eFadeTime:= SEL(bUseGlobalFadeTimeSettings, eFadeTime, eGlobalFadeTime), 
			eFadeRate:= eFadeRate, 
			uiBlinkTi:= nSec_BlinkTi, 
			uiOffDly:= nSec_OffDly, 
			uiPollActLgtLvl:= nSec_PollActLgtLvl, 
			bReInit:= bSec_ReInit, 
			nCycleTimeInMS:= nCycleTimeInMS,
			stLgtCmd:= stLgtCmd_Sec, 
			DALI_LINE_NUM:= DALI_LINE_NUM, 
			fActlLgtLvl=> fActlLgtLvl_Sec, 
			byActlLgtLvl=> byActlLgtLvl_Sec, 
			bLgt=> bLgt_Sec, 
			fActlMinCtrlVal=> fSec_ActlMinCtrlVal, 
			bMinCtrlValRchd=> bSec_MinCtrlValRchd, 
			fActlMaxCtrlVal=> fSec_ActlMaxCtrlVal, 
			bMaxCtrlValRchd=> bSec_MaxCtrlValRchd, 
			fRstVal=>fSec_RstVal, 
			eActlFadeTime=> eSec_ActlFadeTime, 
			eActlFadeRate=> eSec_ActlFadeRate, 
			byPhysMinVal=> nSec_PhysMinVal, 
			byActlMinCtrlVal=> nSec_ActlMinCtrlVal, 
			byActlMaxCtrlVal=> nSec_ActlMaxCtrlVal, 
			bInitDevice=> bSec_InitDevice, 
			bBlinkSeqStarted=> bSec_BlinkSeqStarted, 
			bActionBusy=> bSec_ActionBusy, 
			bErr=> bSec_Err, 
			nErrorId=> nSec_ErrId, 
			byDALIDevSta=> nSec_DALIDevSta);

	END_IF
END_IF
END_METHOD

METHOD M_SuplBallast : BOOL
VAR_INPUT
	byShrtAdr_Supl						: BYTE ;			
	byGrpAdr_Supl						: BYTE ;		
	eMod_Supl							: E_DALIAddressType ;		
	stLgtCmd_Supl						: ST_LgtCmd;	(*Kommandostruktur // command-structure*)
	DALI_LINE_NUM						: BYTE ;	(*DALI-Linie//DALI-line*)
	bUseGlobalFadeTimeSettings			: BOOL := TRUE;
	bReInit								: BOOL;	(*Restart Init-Routine*)
	bTurnOff							: BOOL;	(*Start ramp to 0%*)	
	ipCommunication						: Tc3_DALI.I_DALICommunication;
END_VAR

fbLgtActr_Supl.ipDALICommunication:= ipCommunication;


IF (ipCommunication <> 0) AND (DALI_LINE_NUM <> 0) THEN

	IF eMod_Supl = E_DALIAddressType.Group THEN	
		IF g_arrDiagnosisRunOnce[DALI_LINE_NUM] THEN
			fbMasterSelectorSupl(	
				bErrFromBallastFB:=fbLgtActr_Supl.bErr , 
				byGrpAdr:= byGrpAdr_Supl, 
				DALI_LINE_NUM:= DALI_LINE_NUM, 
				nMasterUnitID=> byShrtAdr_Supl, 
				stGroupSorter:= GVL_DALI.g_arrAddrInGroups[DALI_LINE_NUM]);
		END_IF
	END_IF		

	IF g_arrDiagnosisRunOnce[DALI_LINE_NUM] THEN	

		fbLgtActr_Supl(		
			byShrtAdr:= byShrtAdr_Supl, 
			byGrpAdr:= byGrpAdr_Supl, 
			eMod:= eMod_Supl, 
			fSttupCtrlVal:= stLgtCmd_Supl.fSetCtrlValDct, 
			fMinCtrlVal:= fSupl_MinCtrlVal, 
			fMaxCtrlVal:= fSupl_MaxCtrlVal, 
			fLgtOffset:= fSupl_LgtOffset, 
			eFadeTime:= SEL(bUseGlobalFadeTimeSettings, eFadeTime, eGlobalFadeTime), 
			eFadeRate:= eFadeRate, 
			uiBlinkTi:= nSupl_BlinkTi, 
			uiOffDly:= nSupl_OffDly, 
			uiPollActLgtLvl:= nSupl_PollActLgtLvl, 
			bReInit:= bSupl_ReInit, 
			nCycleTimeInMS:= nCycleTimeInMS,
			stLgtCmd:= stLgtCmd_Supl, 
			DALI_LINE_NUM:= DALI_LINE_NUM, 
			fActlLgtLvl=> fActlLgtLvl_Supl, 
			byActlLgtLvl=> byActlLgtLvl_Supl, 
			bLgt=> bLgt_Supl, 
			fActlMinCtrlVal=> fSupl_ActlMinCtrlVal, 
			bMinCtrlValRchd=> bSupl_MinCtrlValRchd, 
			fActlMaxCtrlVal=> fSupl_ActlMaxCtrlVal, 
			bMaxCtrlValRchd=> bSupl_MaxCtrlValRchd, 
			fRstVal=>fSupl_RstVal, 
			eActlFadeTime=> eSupl_ActlFadeTime, 
			eActlFadeRate=> eSupl_ActlFadeRate, 
			byPhysMinVal=> nSupl_PhysMinVal, 
			byActlMinCtrlVal=> nSupl_ActlMinCtrlVal, 
			byActlMaxCtrlVal=> nSupl_ActlMaxCtrlVal, 
			bInitDevice=> bSupl_InitDevice, 
			bBlinkSeqStarted=> bSupl_BlinkSeqStarted, 
			bActionBusy=> bSupl_ActionBusy, 
			bErr=> bSupl_Err, 
			nErrorId=> nSupl_ErrId, 
			byDALIDevSta=> nSupl_DALIDevSta);

	END_IF
END_IF
END_METHOD

END_FUNCTION_BLOCK

// POUs/DALI/Ballast/FB_MasterSelector
FUNCTION_BLOCK FB_MasterSelector
VAR_INPUT
	bErrFromBallastFB 	: BOOL;
	byGrpAdr			: BYTE;
	DALI_LINE_NUM 		: BYTE;
END_VAR
VAR_OUTPUT
	nMasterUnitID		: BYTE;
END_VAR
VAR
	nSelectIdx : INT;
	fbR_Trig : R_TRIG;
END_VAR
VAR_IN_OUT
	stGroupSorter: ST_GroupSort;
END_VAR



fbR_Trig(CLK:= bErrFromBallastFB);

IF fbR_Trig.Q THEN
	IF (nSelectIdx > 63)  OR (stGroupSorter.arrAddressesInEachGroup[byGrpAdr, nSelectIdx] = 255 )THEN
		nSelectIdx := 0;
	END_IF
	nSelectIdx:= nSelectIdx +1;
END_IF

nMasterUnitID:= stGroupSorter.arrAddressesInEachGroup[byGrpAdr, (nSelectIdx - 1)];

END_FUNCTION_BLOCK

// POUs/DALI/Ballast/FB_Light_SingleBallast
FUNCTION_BLOCK FB_Light_SingleBallast 
VAR_OUTPUT
	bLgt								: BOOL;	(*Light is either on or off*)
	fActlLgtLvl							: REAL;(*Actual light-level in %*)
	byActlLgtLvl						: BYTE;	(*Actual light-level in 0..254*)
	bError		 						: BOOL;
	nError		 						: UINT;	

END_VAR
VAR_INPUT CONSTANT
	nCycleTimeInMS						: UDINT;
END_VAR
VAR

//Global settings for both groups

	eFadeTime							: E_DALIFadeTime:= E_DALIFadeTime.T02000ms;	
	eFadeRate							: E_DALIFadeRate:= E_DALIFadeRate.N063StepsPerSec;		

//Primary group of lamps
	fbLgtActr							: FB_DALILgtActr_EX;		
// Input parameter for Prim row							

	fMinCtrlVal					: REAL := 0;	(*Minimum light-value in %*)				
	fMaxCtrlVal					: REAL := 100;	(*Maximum light-value in %*)				
	fLgtOffset						: REAL := 0;	(*Light-offset-value in %*)				
	nBlinkTi						: UINT := 0;	(*Blinking-sequence Off-pulse in s*)			
	nOffDly						: UINT := 0;	(*Blinking-sequence On-Time after Off-pulse in s*)			
	nPollActLgtLvl					: UINT := 30;	(*Polling-interval light-value/statusbyte*)					
	bReInit						: BOOL;			(*Restart Init-Routine*)	
// Status variables for Primdow row							
	fActlMinCtrlVal				: REAL;	(*Currently programmed min-value in %*)			
	bMinCtrlValRchd				: BOOL;	(*Min-value reached*)			
	fActlMaxCtrlVal				: REAL;	(*Currently programmed max-value in %*)			
	bMaxCtrlValRchd				: BOOL;	(*Max-value reached*)			
	fRstVal						: REAL;	(*Actual reset-value in %*)			
	eActlFadeTime					: E_DALIFadeTime;	(*Currently programmed fade-rate*)			
	eActlFadeRate					: E_DALIFadeRate;	(*Currently programmed fade-rate*)			
	nPhysMinVal					: BYTE;	(*phys. Min-Value in 0..254*)			
	nActlMinCtrlVal				: BYTE;	(*Currently programmed min-value in 0..254*)			
	nActlMaxCtrlVal				: BYTE;	(*Currently programmed max-value in 0..254*)			
	bInitDevice					: BOOL;	(*Init-routine*)			
	bBlinkSeqStarted				: BOOL;	(*Blinking-sequence started*)			
	bActionBusy					: BOOL;	(*DALI-command is being executed*)			
	bErr							: BOOL;	(*Module in error-state*)			
	nErrId							: UDINT;	(*ErrorId*)			
	nDALIDevSta					: BYTE;	(*DALI-Statusbyte*)			
	fbMasterSelectorPrim				: FB_MasterSelector;
END_VAR

METHOD M_Ballast : BOOL
VAR_INPUT
	byShrtAdr							: BYTE:=1;	
	byGrpAdr							: BYTE := 3;	
	eMod								: E_DALIAddressType := E_DALIADDRESSTYPE.Group;
	stLgtCmd							: ST_LgtCmd;	(*Kommandostruktur // command-structure*)
	DALI_LINE_NUM						: BYTE ;	(*DALI-Linie//DALI-line*)
	bUseGlobalFadeTimeSettings			: BOOL := TRUE;
	bReInit								: BOOL;	(*Restart Init-Routine*)
	bTurnOff							: BOOL;	(*Start ramp to 0%*)	
	ipCommunication						: Tc3_DALI.I_DALICommunication;
END_VAR

VAR
END_VAR

fbLgtActr.ipDALICommunication:= ipCommunication;

IF (ipCommunication <> 0) AND (DALI_LINE_NUM <> 0) THEN

	IF eMod = E_DALIAddressType.Group THEN
		IF g_arrDiagnosisRunOnce[DALI_LINE_NUM] THEN
			fbMasterSelectorPrim(
				bErrFromBallastFB:=fbLgtActr.bErr , 
				byGrpAdr:= byGrpAdr, 
				DALI_LINE_NUM:= DALI_LINE_NUM, 
				nMasterUnitID=> byShrtAdr, 
				stGroupSorter:= GVL_DALI.g_arrAddrInGroups[DALI_LINE_NUM]);
		END_IF		
	END_IF
	

(* For checking which task the FB are called*)
	IF g_arrDiagnosisRunOnce[DALI_LINE_NUM] THEN
		fbLgtActr(	
			byShrtAdr:= byShrtAdr, 
			byGrpAdr:= byGrpAdr, 
			eMod:= eMod, 
			fSttupCtrlVal:= stLgtCmd.fSetCtrlValDct, 
			fMinCtrlVal:= fMinCtrlVal, 
			fMaxCtrlVal:= fMaxCtrlVal, 
			fLgtOffset:= fLgtOffset, 
			eFadeTime:= SEL(bUseGlobalFadeTimeSettings, eFadeTime, eGlobalFadeTime), 
			eFadeRate:= eFadeRate, 
			uiBlinkTi:= nBlinkTi, 
			uiOffDly:= nOffDly, 
			uiPollActLgtLvl:= nPollActLgtLvl, 
			bReInit:= bReInit, 
			nCycleTimeInMS:= nCycleTimeInMS,
			stLgtCmd:= stLgtCmd, 
			DALI_LINE_NUM:= DALI_LINE_NUM, 
			fActlLgtLvl=> fActlLgtLvl, 
			byActlLgtLvl=> byActlLgtLvl, 
			bLgt=> bLgt, 
			fActlMinCtrlVal=> fActlMinCtrlVal, 
			bMinCtrlValRchd=> bMinCtrlValRchd, 
			fActlMaxCtrlVal=> fActlMaxCtrlVal, 
			bMaxCtrlValRchd=> bMaxCtrlValRchd, 
			fRstVal=>fRstVal, 
			eActlFadeTime=> eActlFadeTime, 
			eActlFadeRate=> eActlFadeRate, 
			byPhysMinVal=> nPhysMinVal, 
			byActlMinCtrlVal=> nActlMinCtrlVal, 
			byActlMaxCtrlVal=> nActlMaxCtrlVal, 
			bInitDevice=> bInitDevice, 
			bBlinkSeqStarted=> bBlinkSeqStarted, 
			bActionBusy=> bActionBusy, 
			bErr=> bErr, 
			nErrorId=> nErrId, 
			byDALIDevSta=> nDALIDevSta);
	END_IF

END_IF
END_METHOD

END_FUNCTION_BLOCK

// POUs/DALI/Color (DT8)/F_iColorMix
FUNCTION F_iColorMix : dint
VAR_INPUT
	nR, nG, nB : BYTE;
END_VAR
VAR
	pOut : POINTER TO array [0..3] of BYTE;

	nInternR : BYTE;
	nInternG : BYTE;
	nInternB : BYTE;
END_VAR


nInternR := nR;
nInternG := nG;
nInternB := nB;

pOut := ADR(F_iColorMix);

pOut^[0]:= nInternB;
pOut^[1]:= nInternG;
pOut^[2]:= nInternR;

END_FUNCTION

// POUs/DALI/Color (DT8)/FB_DALI_RGBWAFLight
FUNCTION_BLOCK FB_DALI_RGBWAFLight
VAR_INPUT
	bEnable 					: BOOL;
	bSetColor					: BOOL;
	bReadActualTC 				: BOOL;
	nTemporaryRedDimlevel   	: BYTE;
	nTemporaryGreenDimlevel 	: BYTE;
	nTemporaryBlueDimlevel  	: BYTE;
	nTemporaryWhiteDimlevel   	: BYTE;
	nTemporaryAmberDimlevel 	: BYTE;
	nTemporaryFreeColorDimlevel : BYTE;
	byShrtAdr					: BYTE;
	byGrpAdr					: BYTE;
	eAddressType				: Tc3_DALI.E_DALIAddressType;
	eCommandPriority			: Tc3_DALI.E_DALICommandPriority;

	nTemporaryRGBWAFControl		: BYTE; (*	Bit 0 	Output channel 0 / red
										Bit 1 	Output channel 1 / green
										Bit 2 	Output channel 2 / blue
										Bit 3 	Output channel 3 / white
										Bit 4 	Output channel 4 / amber
										Bit 5 	Output channel 5 / free selectable colour
										Bit 6 - 7 	00 = channel control
													01 = colour control
													10 = standardised colour control
													11 = reserved*)
	nDaliLine							: 	INT:=1;
END_VAR
VAR_OUTPUT
	bBusy								: BOOL;
	bError								: BOOL;
	nErrorID							: UDINT;
	iStepBeforeError					: INT;
	nActualRedValue						: BYTE;
	nActualGreenValue					: BYTE;
	nActualBlueValue					: BYTE;
	nActualWhiteValue					: BYTE;
	nActualAmberValue					: BYTE;
	nActualFreeColorValue				: BYTE;
END_VAR
VAR
	
	ipCommunication						:	I_DALICommunication;
	ipCommunicationPreset				:	I_DALICommunication;

	fbDALI209SetTemporaryRGBDimlevel	: FB_DALI209SetTemporaryRGBDimlevel(0); 
	fbDALI209SetTemporaryWAFDimlevel	: FB_DALI209SetTemporaryWAFDimlevel(0) ;
	fbDALI209SetTemporaryRGBWAFControl	: FB_DALI209SetTemporaryRGBWAFControl(0) ;
	fbDALI209QueryColourValueRed		: Tc3_DALI.FB_DALI209QueryColourValue(0);
	fbDALI209QueryColourValueGreen		: Tc3_DALI.FB_DALI209QueryColourValue(0);
	fbDALI209QueryColourValueBlue		: Tc3_DALI.FB_DALI209QueryColourValue(0);
	fbDALI209QueryColourValueWhite		: Tc3_DALI.FB_DALI209QueryColourValue(0);
	fbDALI209QueryColourValueAmber		: Tc3_DALI.FB_DALI209QueryColourValue(0);
	fbDALI209QueryColourValueFree		: Tc3_DALI.FB_DALI209QueryColourValue(0);

	fbDALI209Activate					: Tc3_DALI.FB_DALI209Activate(0);

	nStep				: INT;
	byAddr 				: BYTE;
	eAddrType			: Tc3_DALI.E_DALIAddressType;
	fbTimeOut_TON		: TON;		(* Timer *)
	fbRun_Color_RTRIG 	: R_TRIG;
	fbCycleReadTC_TON	: TON;
	bReadTC				: BOOL:=TRUE;
	bInit				: BOOL ;
	bInitColor			: BOOL ;
	nReadBackValueAddr	: BYTE;
	bRunColorWriteCycle	: BOOL;
	bActionBusy			: BOOL;
	bStart				: BOOL;
	fbDTBlockTimer		: TON;
	fbColorCheck		: TON;
END_VAR


{region "initialize the outputs"}
IF (NOT bInit) THEN
	THIS^.TrySetCommunication();		 
	bBusy := TRUE;
	nErrorId := 0;
	bError := FALSE;
	bInit := TRUE;
END_IF
{endregion}


{region "check parameters"}
IF (ipCommunication = 0) OR (ipCommunication<>ipCommunicationPreset) THEN
	bError := TRUE;
	nErrorId := TC_EVENTS.TcDALIEventClass.TheInterfaceToTheCommunicationBufferIsNotInitialized.nEventId;
	nStep := 0;
 	bInit := FALSE;
	bInitColor:= FALSE;
	RETURN;
END_IF
IF ((eAddressType <> E_DALIAddressType.Short) AND (eAddressType <> E_DALIAddressType.Group) AND (eAddressType <> E_DALIAddressType.Broadcast) AND (eAddressType <> E_DALIAddressType.BroadcastUnaddr)) THEN
	bError := TRUE;
	nErrorId := TC_EVENTS.TcDALIEventClass.ParameterAddressTypeLiesOutsideOfTheValidRange.nEventId;
	nStep := 0;
END_IF
IF ((eAddressType = E_DALIAddressType.Short) AND (byShrtAdr > 63)) THEN
	bError := TRUE;
	nErrorId := TC_EVENTS.TcDALIEventClass.ParameterAddressIsAShortAddressAndLiesOutsideOfTheValidRange.nEventId;
	nStep := 0;
END_IF
IF ((eAddressType = E_DALIAddressType.Group) AND (byGrpAdr > 15)) THEN
	bError := TRUE;
	nErrorId := TC_EVENTS.TcDALIEventClass.ParameterAddressIsAGroupAddressAndLiesOutsideOfTheValidRange.nEventId;
	nStep := 0;
END_IF
IF (byShrtAdr > 63) THEN
	bError := TRUE;
	nErrorId := 16#8000; // custom error code: Parameter byShrtAdr lies outside of the valid range
	nStep := 0;
END_IF
	
IF (byGrpAdr > 15) THEN
	bError := TRUE;
	nErrorId := 16#8001; // custom error code: Parameter byGrpAdr lies outside of the valid range
	nStep := 0;
END_IF
{endregion}


CASE nStep OF


0: //Check if enable are TRUE

	IF bEnable THEN
		nStep := 1;
	END_IF 

	bBusy := FALSE;
	bStart := FALSE;
	fbDALI209QueryColourValueRed(bStart:= FALSE);
	fbDALI209QueryColourValueGreen(bStart:= FALSE);
	fbDALI209QueryColourValueBlue(bStart:= FALSE);
	fbDALI209QueryColourValueAmber(bStart:= FALSE);
	fbDALI209QueryColourValueWhite(bStart:= FALSE);
	fbDALI209QueryColourValueFree(bStart:= FALSE);		
	fbDALI209SetTemporaryRGBDimlevel(bStart:= FALSE);
	fbDALI209SetTemporaryWAFDimlevel(bStart:= FALSE);
	fbDALI209SetTemporaryRGBWAFControl(bStart:= FALSE);	
1: (*Idle*)

	IF NOT bBusy THEN
		fbRun_Color_RTRIG(CLK:=bSetColor, Q=> );
		IF fbRun_Color_RTRIG.Q THEN
			bRunColorWriteCycle:= TRUE;
		END_IF
	
		fbCycleReadTC_TON(IN:= bReadActualTC , PT:=T#1S , Q=> , ET=> );
	
		IF NOT bInitColor AND ((nActualRedValue = 0) AND (nActualGreenValue = 0) AND (nActualBlueValue = 0) AND (nActualWhiteValue = 0) AND (nActualAmberValue = 0))THEN
			bRunColorWriteCycle:=TRUE;
		END_IF

	//Check for correct color in ballast 
	fbColorCheck(IN:= NOT fbColorCheck.Q , PT:= T#2S, Q=> , ET=> );	
	IF fbColorCheck.Q THEN
		IF nTemporaryRedDimlevel <> nActualRedValue OR
			nTemporaryGreenDimlevel <> nActualGreenValue OR
				nTemporaryBlueDimlevel <> nActualBlueValue OR
					nTemporaryWhiteDimlevel <> nActualWhiteValue OR
						nTemporaryAmberDimlevel <> nActualAmberValue THEN
								bRunColorWriteCycle:=TRUE;			
		END_IF
	END_IF

	
		IF  bRunColorWriteCycle AND NOT GVL_DALI.arrbBlockDTR[nDaliLine] THEN
			bBusy:= TRUE;
			A_ResetRoutine();
			nStep:= 10;
			nErrorID:= 0;
			iStepBeforeError:= 0;	
			GVL_DALI.arrbBlockDTR[nDaliLine]:= TRUE;
		END_IF
		
		IF fbCycleReadTC_TON.Q THEN
			bBusy:= TRUE;
			bReadTC:= FALSE;
			A_ResetRoutine();
			nStep:= 100;
			nErrorID:= 0;
			iStepBeforeError:= 0;
		END_IF
	END_IF
	
(* - - - - - - - - - - - - - - - - - - - - - - - - *)
10:(*Set color temperatur to ballast*)
	bStart:= TRUE;
	A_DALICmdTemporaryRGBDimlevel();
	IF NOT bActionBusy	THEN
		IF bError	THEN
			GVL_DALI.arrbBlockDTR[nDaliLine]:= FALSE;
			nStep:= 0;
		ELSE
			bStart := FALSE;
			nStep:= 11;
		END_IF
	END_IF

11, 13, 15: (* Activate the color temp send to ballast*)

	A_DALICmdActivate_DT8();
	
	IF NOT bActionBusy	THEN
		IF bError	THEN
			GVL_DALI.arrbBlockDTR[nDaliLine]:= FALSE;
			nStep:= 0;
		ELSE
			bStart := FALSE;
			IF nStep = 11 THEN
				nStep:= 12;	
			ELSIF nStep = 13 THEN
				nStep:= 14;
			ELSIF nStep = 15 THEN
				nStep:= 100;	
			END_IF
		END_IF
	END_IF	



12: (* Set WAF Values to ballast*)

	A_DALICmdTemporaryWAFDimlevel();
	IF NOT bActionBusy	THEN
		nStep:= 13;
	END_IF

	
14: (* Set color Control to ballast*)

	A_DALICmdTemporaryRGBWAFControl();
	IF NOT bActionBusy	THEN
		nStep:= 15;
	END_IF


100: (*Read back current Red color*)

	A_DALIQueryColourValueRed();
	IF NOT bActionBusy	THEN
		nStep:= 101;
	END_IF
	
	

101: (*Read back current Green color*)

		A_DALIQueryColourValueGreen();
	IF NOT bActionBusy	THEN
		nStep:= 102;
	END_IF

102: (*Read back current Blue color*)
	A_DALIQueryColourValueBlue();
	IF NOT bActionBusy	THEN
		nStep:= 103;
	END_IF

103: (*Read back current White color*)

	A_DALIQueryColourValueWhite();
	IF NOT bActionBusy	THEN
		nStep:= 104;
	END_IF


104: (*Read back current Amber color*)

	A_DALIQueryColourValueAmber();
	IF NOT bActionBusy	THEN
		nStep:= 105;
	END_IF


105: (*Read back current Free color*)

	A_DALIQueryColourValueFreeColor();
	IF NOT bActionBusy	THEN
		nStep:= 888;
	END_IF

		
888: (*Done step*)
	bBusy:= FALSE;
	nStep:=0;
	nErrorID:= 0;
	iStepBeforeError:= 0;
	bRunColorWriteCycle:= FALSE;
	bInitColor:= TRUE;
	GVL_DALI.arrbBlockDTR[nDaliLine]:= FALSE;
ELSE
	nStep := 0;
END_CASE

//Checking if this FB blocks DT_Telegrams for other ballast

fbDTBlockTimer(IN:=GVL_DALI.arrbBlockDTR[nDaliLine] AND (nStep > 0) AND NOT fbDTBlockTimer.Q , PT:= T#20S , Q=> , ET=> );

IF fbDTBlockTimer.Q THEN
	nStep := 0;
	GVL_DALI.arrbBlockDTR[nDaliLine]:= FALSE;
END_IF

	nActualRedValue := UINT_TO_BYTE((fbDALI209QueryColourValueRed.nColourValue / 255) -1);
	nActualGreenValue := UINT_TO_BYTE((fbDALI209QueryColourValueGreen.nColourValue / 255) -1);
	nActualBlueValue := UINT_TO_BYTE((fbDALI209QueryColourValueBlue.nColourValue / 255) -1);
	nActualWhiteValue := UINT_TO_BYTE((fbDALI209QueryColourValueWhite.nColourValue / 255) -1);
	nActualAmberValue := UINT_TO_BYTE((fbDALI209QueryColourValueAmber.nColourValue / 255) -1);
	nActualFreeColorValue := UINT_TO_BYTE((fbDALI209QueryColourValueFree.nColourValue / 255) -1);

ACTION A_DALICmdActivate_DT8:
IF eAddressType= E_DALIAddressType.Group THEN
	byAddr		:= byGrpAdr;
	eAddrType	:= E_DALIAddressType.Group;
END_IF

IF eAddressType= E_DALIAddressType.Short THEN
	byAddr		:= byShrtAdr;
	eAddrType	:= E_DALIAddressType.Short;
END_IF

	bActionBusy	:= TRUE;

	fbDALI209Activate(
		bError=> , 
		ipResultMessage=> , 
		bStart:= TRUE, 
		nAddress:= byAddr , 
		eAddressType:= eAddressType, 
		eCommandPriority:=eCommandPriority ,
		bBusy=> );
	

	IF (NOT fbDALI209Activate.bBusy) THEN
		IF fbDALI209Activate.bError THEN
			bError := TRUE;
			nErrorId := fbDALI209Activate.ipResultMessage.nEventId;
		END_IF
		bActionBusy		:= FALSE;
		fbDALI209Activate(bStart:= FALSE);
	END_IF
END_ACTION

ACTION A_DALICmdTemporaryRGBDimlevel:
IF eAddressType= E_DALIAddressType.Group THEN
	byAddr		:= byGrpAdr;
	eAddrType	:= E_DALIAddressType.Group;
END_IF

IF eAddressType= E_DALIAddressType.Short THEN
	byAddr		:= byShrtAdr;
	eAddrType	:= E_DALIAddressType.Short;
END_IF

	bActionBusy	:= TRUE;

	fbDALI209SetTemporaryRGBDimlevel(
		bError=> , 
		ipResultMessage=> , 
		bStart:= TRUE, 
		nAddress:= byAddr , 
		eAddressType:= eAddressType, 
		eCommandPriority:=eCommandPriority , 
		bBusy=> , 
		nTemporaryRedDimlevel:= nTemporaryRedDimlevel, 
		nTemporaryGreenDimlevel:= nTemporaryGreenDimlevel , 
		nTemporaryBlueDimlevel:= nTemporaryBlueDimlevel );
	
	
	
	IF (NOT fbDALI209SetTemporaryRGBDimlevel.bBusy) THEN
		IF fbDALI209SetTemporaryRGBDimlevel.bError THEN
			bError := TRUE;
			nErrorId := fbDALI209SetTemporaryRGBDimlevel.ipResultMessage.nEventId;
		END_IF
		bActionBusy		:= FALSE;
		fbDALI209SetTemporaryRGBDimlevel(bStart:= FALSE);
	END_IF
END_ACTION

ACTION A_DALICmdTemporaryRGBWAFControl:
IF eAddressType= E_DALIAddressType.Group THEN
	byAddr		:= byGrpAdr;
	eAddrType	:= E_DALIAddressType.Group;
END_IF

IF eAddressType= E_DALIAddressType.Short THEN
	byAddr		:= byShrtAdr;
	eAddrType	:= E_DALIAddressType.Short;
END_IF

	bActionBusy	:= TRUE;

	fbDALI209SetTemporaryRGBWAFControl(
		bError=> , 
		ipResultMessage=> , 
		bStart:= TRUE, 
		nAddress:= byAddr , 
		eAddressType:= eAddressType, 
		eCommandPriority:=eCommandPriority , 
		bBusy=> , 
		nTemporaryRGBWAFControl:= nTemporaryRGBWAFControl);
	

	
	IF (NOT fbDALI209SetTemporaryRGBWAFControl.bBusy) THEN
		IF fbDALI209SetTemporaryRGBWAFControl.bError THEN
			bError := TRUE;
			nErrorId := fbDALI209SetTemporaryRGBWAFControl.ipResultMessage.nEventId;
		END_IF
		bActionBusy		:= FALSE;
		fbDALI209SetTemporaryRGBWAFControl(bStart:= FALSE);
	END_IF
END_ACTION

ACTION A_DALICmdTemporaryWAFDimlevel:
IF eAddressType= E_DALIAddressType.Group THEN
	byAddr		:= byGrpAdr;
	eAddrType	:= E_DALIAddressType.Group;
END_IF

IF eAddressType= E_DALIAddressType.Short THEN
	byAddr		:= byShrtAdr;
	eAddrType	:= E_DALIAddressType.Short;
END_IF

	bActionBusy	:= TRUE;

	fbDALI209SetTemporaryWAFDimlevel(
		bError=> , 
		ipResultMessage=> , 
		bStart:= TRUE, 
		nAddress:= byAddr , 
		eAddressType:= eAddressType, 
		eCommandPriority:=eCommandPriority, 
		bBusy=> , 
		nTemporaryWhiteDimlevel:= nTemporaryWhiteDimlevel, 
		nTemporaryAmberDimlevel:= nTemporaryAmberDimlevel, 
		nTemporaryFreecolourDimlevel:= nTemporaryFreeColorDimlevel);
	

	
	IF (NOT fbDALI209SetTemporaryWAFDimlevel.bBusy) THEN
		IF fbDALI209SetTemporaryWAFDimlevel.bError THEN
			bError := TRUE;
			nErrorId := fbDALI209SetTemporaryWAFDimlevel.ipResultMessage.nEventId;
		END_IF
		bActionBusy		:= FALSE;
		fbDALI209SetTemporaryWAFDimlevel(bStart:= FALSE);
	END_IF
END_ACTION

ACTION A_DALIQueryColourValueAmber:

	byAddr:= byShrtAdr;

	bActionBusy	:= TRUE;


	fbDALI209QueryColourValueAmber(
		bError=> , 
		ipResultMessage=> , 
		bStart:= TRUE , 
		nAddress:=byAddr , 
		eAddressType:= Tc3_DALI.E_DALIAddressType.Short, 
		eCommandPriority:= Tc3_DALI.E_DALICommandPriority.Low, 
		bBusy=> , 
		eColourValue:= Tc3_DALI.E_DALIColourValue.AmberDimlevel , 
		nColourValue=> );	
	

	IF (NOT fbDALI209QueryColourValueAmber.bBusy) THEN
		IF fbDALI209QueryColourValueAmber.bError THEN
			bError := TRUE;
			nErrorId := fbDALI209QueryColourValueAmber.ipResultMessage.nEventId;
		END_IF
		bActionBusy		:= FALSE;
		fbDALI209QueryColourValueAmber(bStart:= FALSE);
	END_IF
END_ACTION

ACTION A_DALIQueryColourValueBlue:

	byAddr:= byShrtAdr;

	bActionBusy	:= TRUE;


	fbDALI209QueryColourValueBlue(
		bError=> , 
		ipResultMessage=> , 
		bStart:= TRUE , 
		nAddress:=byAddr , 
		eAddressType:= Tc3_DALI.E_DALIAddressType.Short, 
		eCommandPriority:= Tc3_DALI.E_DALICommandPriority.Low, 
		bBusy=> , 
		eColourValue:= Tc3_DALI.E_DALIColourValue.BlueDimlevel , 
		nColourValue=> );	
	

	IF (NOT fbDALI209QueryColourValueBlue.bBusy) THEN
		IF fbDALI209QueryColourValueBlue.bError THEN
			bError := TRUE;
			nErrorId := fbDALI209QueryColourValueBlue.ipResultMessage.nEventId;
		END_IF
		bActionBusy		:= FALSE;
		fbDALI209QueryColourValueBlue(bStart:= FALSE);
	END_IF
END_ACTION

ACTION A_DALIQueryColourValueFreeColor:

	byAddr:= byShrtAdr;

	bActionBusy	:= TRUE;


	fbDALI209QueryColourValueFree(
		bError=> , 
		ipResultMessage=> , 
		bStart:= TRUE , 
		nAddress:=byAddr , 
		eAddressType:= Tc3_DALI.E_DALIAddressType.Short, 
		eCommandPriority:= Tc3_DALI.E_DALICommandPriority.Low, 
		bBusy=> , 
		eColourValue:= Tc3_DALI.E_DALIColourValue.FreecolourDimlevel , 
		nColourValue=> );	
	

	IF (NOT fbDALI209QueryColourValueFree.bBusy) THEN
		IF fbDALI209QueryColourValueFree.bError THEN
			bError := TRUE;
			nErrorId := fbDALI209QueryColourValueFree.ipResultMessage.nEventId;
		END_IF
		bActionBusy		:= FALSE;
		fbDALI209QueryColourValueFree(bStart:= FALSE);
	END_IF
END_ACTION

ACTION A_DALIQueryColourValueGreen:

	byAddr:= byShrtAdr;

	bActionBusy	:= TRUE;


	fbDALI209QueryColourValueGreen(
		bError=> , 
		ipResultMessage=> , 
		bStart:= TRUE , 
		nAddress:=byAddr , 
		eAddressType:= Tc3_DALI.E_DALIAddressType.Short, 
		eCommandPriority:= Tc3_DALI.E_DALICommandPriority.Low, 
		bBusy=> , 
		eColourValue:= Tc3_DALI.E_DALIColourValue.GreenDimlevel , 
		nColourValue=> );	
	

	IF (NOT fbDALI209QueryColourValueGreen.bBusy) THEN
		IF fbDALI209QueryColourValueGreen.bError THEN
			bError := TRUE;
			nErrorId := fbDALI209QueryColourValueGreen.ipResultMessage.nEventId;
		END_IF
		bActionBusy		:= FALSE;
		fbDALI209QueryColourValueGreen(bStart:= FALSE);
	END_IF
END_ACTION

ACTION A_DALIQueryColourValueRed:

	byAddr:= byShrtAdr;

	bActionBusy	:= TRUE;


	fbDALI209QueryColourValueRed(
		bError=> , 
		ipResultMessage=> , 
		bStart:= TRUE , 
		nAddress:=byAddr , 
		eAddressType:= Tc3_DALI.E_DALIAddressType.Short, 
		eCommandPriority:= Tc3_DALI.E_DALICommandPriority.Low, 
		bBusy=> , 
		eColourValue:= Tc3_DALI.E_DALIColourValue.RedDimlevel, 
		nColourValue=> );	
	

	IF (NOT fbDALI209QueryColourValueRed.bBusy) THEN
		IF fbDALI209QueryColourValueRed.bError THEN
			bError := TRUE;
			nErrorId := fbDALI209QueryColourValueRed.ipResultMessage.nEventId;
		END_IF
		bActionBusy		:= FALSE;
		fbDALI209QueryColourValueRed(bStart:= FALSE);
	END_IF
END_ACTION

ACTION A_DALIQueryColourValueWhite:

	byAddr:= byShrtAdr;

	bActionBusy	:= TRUE;


	fbDALI209QueryColourValueWhite(
		bError=> , 
		ipResultMessage=> , 
		bStart:= TRUE , 
		nAddress:=byAddr , 
		eAddressType:= Tc3_DALI.E_DALIAddressType.Short, 
		eCommandPriority:= Tc3_DALI.E_DALICommandPriority.Low, 
		bBusy=> , 
		eColourValue:= Tc3_DALI.E_DALIColourValue.WhiteDimLevel , 
		nColourValue=> );	
	

	IF (NOT fbDALI209QueryColourValueWhite.bBusy) THEN
		IF fbDALI209QueryColourValueWhite.bError THEN
			bError := TRUE;
			nErrorId := fbDALI209QueryColourValueWhite.ipResultMessage.nEventId;
		END_IF
		bActionBusy		:= FALSE;
		fbDALI209QueryColourValueWhite(bStart:= FALSE);
	END_IF
END_ACTION

ACTION A_ResetRoutine:

	bError     	:= FALSE;
	nErrorId	:= 0;

	fbDALI209SetTemporaryRGBDimlevel (bStart:= FALSE);
	fbDALI209SetTemporaryWAFDimlevel (bStart:= FALSE);
	fbDALI209SetTemporaryRGBWAFControl (bStart:= FALSE);
	fbDALI209QueryColourValueRed(bStart:= FALSE);
	fbDALI209QueryColourValueGreen(bStart:= FALSE);
	fbDALI209QueryColourValueBlue(bStart:= FALSE);
	fbDALI209QueryColourValueWhite(bStart:= FALSE);
	fbDALI209QueryColourValueAmber(bStart:= FALSE);
	fbDALI209QueryColourValueFree(bStart:= FALSE);
	fbDALI209Activate(bStart:= FALSE);
END_ACTION

{attribute 'monitoring' := 'call'}
PROPERTY ipDALICommunication : Tc3_DALI.I_DALICommunication
GET
ipDALICommunication := THIS^.ipCommunication;
END_GET
SET
THIS^.ipCommunicationPreset := ipDALICommunication;
END_SET
END_PROPERTY

//| Apply the perset value of IpCommunication if available
//| Return codes:
//|   FALSE: no peset value available
//|   TRUE: has taken the preset value
{attribute 'hide'}
METHOD PRIVATE TrySetCommunication : BOOL
VAR_INPUT
END_VAR
IF ((THIS^.ipCommunication <> THIS^.ipCommunicationPreset) AND (THIS^.ipCommunicationPreset <> 0)) THEN
	THIS^.ipCommunication := THIS^.ipCommunicationPreset;
	THIS^.fbDALI209SetTemporaryRGBDimlevel.ipDALICommunication := THIS^.ipCommunication;
	THIS^.fbDALI209SetTemporaryWAFDimlevel.ipDALICommunication := THIS^.ipCommunication;
	THIS^.fbDALI209SetTemporaryRGBWAFControl.ipDALICommunication := THIS^.ipCommunication;
	THIS^.fbDALI209QueryColourValueRed.ipDALICommunication := THIS^.ipCommunication;
	THIS^.fbDALI209QueryColourValueGreen.ipDALICommunication := THIS^.ipCommunication;
	THIS^.fbDALI209QueryColourValueBlue.ipDALICommunication := THIS^.ipCommunication;
	THIS^.fbDALI209QueryColourValueWhite.ipDALICommunication := THIS^.ipCommunication;	
	THIS^.fbDALI209QueryColourValueAmber.ipDALICommunication := THIS^.ipCommunication;
	THIS^.fbDALI209QueryColourValueFree.ipDALICommunication := THIS^.ipCommunication;	
	THIS^.fbDALI209Activate.ipDALICommunication := THIS^.ipCommunication;

	TrySetCommunication := TRUE;
ELSE
	TrySetCommunication := FALSE;
END_IF
END_METHOD

END_FUNCTION_BLOCK

// POUs/DALI/Color (DT8)/FB_DALI_TcColorLight
FUNCTION_BLOCK FB_DALI_TcColorLight
VAR_INPUT
	bEnable 					: BOOL;
	bSetColor					: BOOL;
	bReadActualTC 				: BOOL;
	fColourTemperatureTc 		: LREAL;
	byShrtAdr					: BYTE;
	byGrpAdr					: BYTE;
	eAddressType				: Tc3_DALI.E_DALIAddressType;
	eCommandPriority			: Tc3_DALI.E_DALICommandPriority;

	nDaliLine							: 	INT:=1;
END_VAR
VAR_OUTPUT
	bBusy								: BOOL;
	bError								: BOOL;
	nErrorID							: UDINT;
	iStepBeforeError					: INT;
	fActualTcColor						: LREAL;
	nActualColorStatus					: BYTE;

END_VAR
VAR
	
	ipCommunication						: I_DALICommunication;
	ipCommunicationPreset				: I_DALICommunication;

	fbDALI209SetColourTemperatureTc		: Tc3_DALI.FB_DALI209SetColourTemperatureTc(0); 
	fbDALI209QueryColourStatus			: Tc3_DALI.FB_DALI209QueryColourStatus(0);
	fbDALI209QueryColourTc				: Tc3_DALI.FB_DALI209QueryColourValue(0);
	fbDALI209Activate					: Tc3_DALI.FB_DALI209Activate(0);

	nStep				: INT;
	byAddr 				: BYTE;
	eAddrType			: Tc3_DALI.E_DALIAddressType;
	fbTimeOut_TON		: TON;		(* Timer *)
	fbRun_Color_RTRIG 	: R_TRIG;
	fbCycleReadTC_TON	: TON;
	bReadTC				: BOOL:=TRUE;
	bInit				: BOOL ;
	bInitColor			: BOOL ;
	nReadBackValueAddr	: BYTE;
	bRunColorWriteCycle	: BOOL;
	bActionBusy			: BOOL;
	bStart				: BOOL;
	fbDTBlockTimer		: TON;
	fbColorCheck		: TON;
END_VAR

{region "initialize the outputs"}
IF (NOT bInit) THEN
	THIS^.TrySetCommunication();		 
	bBusy := TRUE;
	nErrorId := 0;
	bError := FALSE;
	bInit := TRUE;
END_IF
{endregion}


{region "check parameters"}
IF (ipCommunication = 0) OR (ipCommunication<>ipCommunicationPreset) THEN
	bError := TRUE;
	nErrorId := TC_EVENTS.TcDALIEventClass.TheInterfaceToTheCommunicationBufferIsNotInitialized.nEventId;
	nStep := 0;
 	bInit := FALSE;
	bInitColor:= FALSE;
	RETURN;
END_IF
IF ((eAddressType <> E_DALIAddressType.Short) AND (eAddressType <> E_DALIAddressType.Group) AND (eAddressType <> E_DALIAddressType.Broadcast) AND (eAddressType <> E_DALIAddressType.BroadcastUnaddr)) THEN
	bError := TRUE;
	nErrorId := TC_EVENTS.TcDALIEventClass.ParameterAddressTypeLiesOutsideOfTheValidRange.nEventId;
	nStep := 0;
END_IF
IF ((eAddressType = E_DALIAddressType.Short) AND (byShrtAdr > 63)) THEN
	bError := TRUE;
	nErrorId := TC_EVENTS.TcDALIEventClass.ParameterAddressIsAShortAddressAndLiesOutsideOfTheValidRange.nEventId;
	nStep := 0;
END_IF
IF ((eAddressType = E_DALIAddressType.Group) AND (byGrpAdr > 15)) THEN
	bError := TRUE;
	nErrorId := TC_EVENTS.TcDALIEventClass.ParameterAddressIsAGroupAddressAndLiesOutsideOfTheValidRange.nEventId;
	nStep := 0;
END_IF
IF (byShrtAdr > 63) THEN
	bError := TRUE;
	nErrorId := 16#8000; // custom error code: Parameter byShrtAdr lies outside of the valid range
	nStep := 0;
END_IF
	
IF (byGrpAdr > 15) THEN
	bError := TRUE;
	nErrorId := 16#8001; // custom error code: Parameter byGrpAdr lies outside of the valid range
	nStep := 0;
END_IF
{endregion}


CASE nStep OF


0: //Check if enable are TRUE

	IF bEnable THEN
		nStep := 1;
	END_IF 

	bBusy := FALSE;
	bStart := FALSE;
	fbDALI209SetColourTemperatureTc(bStart:= FALSE);
	fbDALI209QueryColourStatus(bStart:= FALSE);
	fbDALI209QueryColourTc(bStart:= FALSE);
	fbDALI209Activate(bStart:= FALSE);
	
1: (*Idle*)

